DATA_BLOCK "InstGetSinaStatus"   // DB15
AUTHOR : Siemens Digital Industries
FAMILY : LAF
NAME : LAF_GetSinaStatus
VERSION : 1.1
// stored: InstanceOfName LAF_GetSinaStatus, InstanceOfType FB
"LAF_GetSinaStatus"
   // VAR_INPUT
   //    enable : Bool;
   // END_VAR
   // VAR_OUTPUT
   //    valid { ExternalWritable := 'False'} : Bool;
   //    busy { ExternalWritable := 'False'} : Bool;
   //    error { ExternalWritable := 'False'} : Bool;
   //    status { ExternalWritable := 'False'} : Word;
   //    diagnostics { ExternalWritable := 'False'} : "LAF_typeDiagnostics";
   //    statusWriteRecord { ExternalVisible := 'False'; ExternalWritable := 'False'} : DWord;
   //    statusReadRecord { ExternalWritable := 'False'} : DWord;
   // END_VAR
   // VAR_IN_OUT
   //    configuration : Array[*] of "LAF_typeDriveDiagConfig";
   //    moduleInterface : "LAF_typeDriveDiagInterfaceHmi";
   // END_VAR
   // VAR
   //    statInternal { ExternalAccessible := 'False'; ExternalVisible := 'False'; ExternalWritable := 'False'} : Struct
   //       enablePrevious : Bool;
   //       valid : Bool;
   //       busy : Bool;
   //       error : Bool;
   //       errorUserCleared : Bool;
   //       errorAutoCleared : Bool;
   //       disablingCompleted : Bool;
   //       diagnostics : "LAF_typeDiagnostics";
   //       emptyDiagnostics : "LAF_typeDiagnostics";
   //    END_STRUCT;
   //    statMainState { ExternalAccessible := 'False'; ExternalVisible := 'False'; ExternalWritable := 'False'} : DInt;
   //    statArrayMin { ExternalAccessible := 'False'; ExternalVisible := 'False'; ExternalWritable := 'False'} : DInt;
   //    statArrayMax { ExternalAccessible := 'False'; ExternalVisible := 'False'; ExternalWritable := 'False'} : DInt;
   //    instWriteRecord { ExternalAccessible := 'False'; ExternalVisible := 'False'; ExternalWritable := 'False'} : WRREC;
   //    instReadRecord { ExternalAccessible := 'False'; ExternalVisible := 'False'; ExternalWritable := 'False'} : RDREC;
   //    statWriteReq { ExternalAccessible := 'False'; ExternalVisible := 'False'; ExternalWritable := 'False'} : Struct
   //       header : Struct
   //          reqRef : Byte;
   //          reqID : Byte;
   //          axis : Byte;
   //          noPara : Byte;
   //       END_STRUCT;
   //       data : Array[0..235] of Byte;
   //    END_STRUCT;
   //    statReadReq { ExternalAccessible := 'False'; ExternalVisible := 'False'; ExternalWritable := 'False'} : Struct
   //       header : Struct
   //          reqRef : Byte;
   //          reqID : Byte;
   //          axis : Byte;
   //          noPara : Byte;
   //       END_STRUCT;
   //       data : Array[0..235] of Byte;
   //    END_STRUCT;
   //    instActTimer { ExternalAccessible := 'False'; ExternalVisible := 'False'; ExternalWritable := 'False'} : IEC_TIMER;
   //    instReqTimer { ExternalAccessible := 'False'; ExternalVisible := 'False'; ExternalWritable := 'False'} : IEC_TIMER;
   //    statDataTransRun { ExternalAccessible := 'False'; ExternalVisible := 'False'; ExternalWritable := 'False'} : Bool;
   //    statWriteReqSet { ExternalAccessible := 'False'; ExternalVisible := 'False'; ExternalWritable := 'False'} : Bool;
   //    statActTimerIn { ExternalAccessible := 'False'; ExternalVisible := 'False'; ExternalWritable := 'False'} : Bool;
   //    statPrevTimeValue { ExternalAccessible := 'False'; ExternalVisible := 'False'; ExternalWritable := 'False'} : Time;
   //    statActTimerValueAct { ExternalAccessible := 'False'; ExternalVisible := 'False'; ExternalWritable := 'False'} : Time;
   //    statActTimerValueReq { ExternalAccessible := 'False'; ExternalVisible := 'False'; ExternalWritable := 'False'} : Time;
   //    statPrevDriveIndex { ExternalAccessible := 'False'; ExternalVisible := 'False'; ExternalWritable := 'False'} : DInt;
   // END_VAR
BEGIN
END_DATA_BLOCK

DATA_BLOCK "InstInterfaceSignals"   // DB39
{ DB_Accessible_From_OPC_UA := 'FALSE' }
AUTHOR : SICAR
FAMILY : Diag
VERSION : 1.0
// stored: DBAccessibleFromOPCUA false, DBAccessibleFromWebserver false, InstanceOfName CallInterfaceSignals, InstanceOfType FB
"CallInterfaceSignals"
BEGIN
   statInterfaceSignalsHmi[1].valueSymbolLeft.freeDescriptionText := WSTRING#'ReelCut To STK30';
   statInterfaceSignalsHmi[2].valueSymbolLeft.freeDescriptionText := WSTRING#'ReelCut to STK40';
   statInterfaceSignalsHmi[3].valueSymbolLeft.freeDescriptionText := WSTRING#'BK01';
   statInterfaceSignalsHmi[4].valueSymbolLeft.freeDescriptionText := WSTRING#'BK02';
   statInterfaceSignalsHmi[5].valueSymbolLeft.freeDescriptionText := WSTRING#'BK03';
   statInterfaceSignalsHmi[6].valueSymbolLeft.freeDescriptionText := WSTRING#'BK04';
   statInterfaceSignalsHmi[7].valueSymbolLeft.freeDescriptionText := WSTRING#'BK05';
   statInterfaceSignalsHmi[8].valueSymbolLeft.freeDescriptionText := WSTRING#'BK06';
   statInterfaceSignalsHmi[9].valueSymbolLeft.freeDescriptionText := WSTRING#'BK07';
   statInterfaceSignalsHmi[10].valueSymbolLeft.freeDescriptionText := WSTRING#'BK08';
   statInterfaceSignalsHmi[11].valueSymbolLeft.freeDescriptionText := WSTRING#'BK09';
   statInterfaceSignalsHmi[12].valueSymbolLeft.freeDescriptionText := WSTRING#'BK10';
   statInterfaceSignalsHmi[13].valueSymbolLeft.freeDescriptionText := WSTRING#'SBK01';
   statInterfaceSignalsHmi[14].valueSymbolLeft.freeDescriptionText := WSTRING#'SBK02';
   statInterfaceSignalsHmi[15].valueSymbolLeft.freeDescriptionText := WSTRING#'SBK03';
   statInterfaceSignalsHmi[16].valueSymbolLeft.freeDescriptionText := WSTRING#'SBK04';
   statInterfaceSignalsHmi[17].valueSymbolLeft.freeDescriptionText := WSTRING#'SBK05';
   statInterfaceSignalsHmi[18].valueSymbolLeft.freeDescriptionText := WSTRING#'SBK06';
   statInterfaceSignalsHmi[19].valueSymbolLeft.freeDescriptionText := WSTRING#'SBK01';
   statInterfaceSignalsHmi[20].valueSymbolLeft.freeDescriptionText := WSTRING#'SBK02';
   statInterfaceSignalsHmi[21].valueSymbolLeft.freeDescriptionText := WSTRING#'SBK03';
   statInterfaceSignalsHmi[22].valueSymbolLeft.freeDescriptionText := WSTRING#'SBK04';
   statInterfaceSignalsHmi[23].valueSymbolLeft.freeDescriptionText := WSTRING#'SBK05';
   statInterfaceSignalsHmi[24].valueSymbolLeft.freeDescriptionText := WSTRING#'SBK06';
   statInterfaceSignalsHmi[25].valueSymbolLeft.freeDescriptionText := WSTRING#'SBK07';
   statInterfaceSignalsHmi[26].valueSymbolLeft.freeDescriptionText := WSTRING#'SBK08';
   statInterfaceSignalsHmi[27].valueSymbolLeft.freeDescriptionText := WSTRING#'SBK09';
   statInterfaceSignalsHmi[28].valueSymbolLeft.freeDescriptionText := WSTRING#'PM01';
   statInterfaceSignalsHmi[29].valueSymbolLeft.freeDescriptionText := WSTRING#'PM02';
   statInterfaceSignalsHmi[30].valueSymbolLeft.freeDescriptionText := WSTRING#'PM03';
   statInterfaceSignalsHmi[31].valueSymbolLeft.freeDescriptionText := WSTRING#'PM04';
   statInterfaceSignalsHmi[37].valueSymbolLeft.freeDescriptionText := WSTRING#'SP501';
   statInterfaceSignalsHmi[38].valueSymbolLeft.freeDescriptionText := WSTRING#'SP502';
   statInterfaceSignalsHmi[39].valueSymbolLeft.freeDescriptionText := WSTRING#'SP503';
   statInterfaceSignalsHmi[40].valueSymbolLeft.freeDescriptionText := WSTRING#'SP504';
   statInterfaceSignalsHmi[41].valueSymbolLeft.freeDescriptionText := WSTRING#'SP505';
   statInterfaceSignalsHmi[42].valueSymbolLeft.freeDescriptionText := WSTRING#'SP506';
   statInterfaceSignalsHmi[43].valueSymbolLeft.freeDescriptionText := WSTRING#'SP507';
   statInterfaceSignalsHmi[44].valueSymbolLeft.freeDescriptionText := WSTRING#'SP508';
   statInterfaceSignalsHmi[45].valueSymbolLeft.freeDescriptionText := WSTRING#'SP509';
   statInterfaceSignalsHmi[46].valueSymbolLeft.freeDescriptionText := WSTRING#'SP510';
   statInterfaceSignalsHmi[47].valueSymbolLeft.freeDescriptionText := WSTRING#'SP511';
   statInterfaceSignalsHmi[48].valueSymbolLeft.freeDescriptionText := WSTRING#'SP512';
   statInterfaceSignalsHmi[1].valueSymbolRight.freeDescriptionText := WSTRING#'ReelCut To STK30';
   statInterfaceSignalsHmi[2].valueSymbolRight.freeDescriptionText := WSTRING#'ReelCut to STK40';
   statInterfaceSignalsHmi[3].valueSymbolRight.freeDescriptionText := WSTRING#'BK01';
   statInterfaceSignalsHmi[4].valueSymbolRight.freeDescriptionText := WSTRING#'BK02';
   statInterfaceSignalsHmi[5].valueSymbolRight.freeDescriptionText := WSTRING#'BK03';
   statInterfaceSignalsHmi[6].valueSymbolRight.freeDescriptionText := WSTRING#'BK04';
   statInterfaceSignalsHmi[7].valueSymbolRight.freeDescriptionText := WSTRING#'BK05';
   statInterfaceSignalsHmi[8].valueSymbolRight.freeDescriptionText := WSTRING#'BK06';
   statInterfaceSignalsHmi[9].valueSymbolRight.freeDescriptionText := WSTRING#'BK07';
   statInterfaceSignalsHmi[10].valueSymbolRight.freeDescriptionText := WSTRING#'BK08';
   statInterfaceSignalsHmi[11].valueSymbolRight.freeDescriptionText := WSTRING#'BK09';
   statInterfaceSignalsHmi[12].valueSymbolRight.freeDescriptionText := WSTRING#'BK10';
   statInterfaceSignalsHmi[13].valueSymbolRight.freeDescriptionText := WSTRING#'SBK01';
   statInterfaceSignalsHmi[14].valueSymbolRight.freeDescriptionText := WSTRING#'SBK02';
   statInterfaceSignalsHmi[15].valueSymbolRight.freeDescriptionText := WSTRING#'SBK03';
   statInterfaceSignalsHmi[16].valueSymbolRight.freeDescriptionText := WSTRING#'SBK04';
   statInterfaceSignalsHmi[17].valueSymbolRight.freeDescriptionText := WSTRING#'SBK05';
   statInterfaceSignalsHmi[18].valueSymbolRight.freeDescriptionText := WSTRING#'SBK06';
   statInterfaceSignalsHmi[19].valueSymbolRight.freeDescriptionText := WSTRING#'SBK01';
   statInterfaceSignalsHmi[20].valueSymbolRight.freeDescriptionText := WSTRING#'SBK02';
   statInterfaceSignalsHmi[21].valueSymbolRight.freeDescriptionText := WSTRING#'SBK03';
   statInterfaceSignalsHmi[22].valueSymbolRight.freeDescriptionText := WSTRING#'SBK04';
   statInterfaceSignalsHmi[23].valueSymbolRight.freeDescriptionText := WSTRING#'SBK05';
   statInterfaceSignalsHmi[24].valueSymbolRight.freeDescriptionText := WSTRING#'SBK06';
   statInterfaceSignalsHmi[25].valueSymbolRight.freeDescriptionText := WSTRING#'SBK07';
   statInterfaceSignalsHmi[26].valueSymbolRight.freeDescriptionText := WSTRING#'SBK08';
   statInterfaceSignalsHmi[27].valueSymbolRight.freeDescriptionText := WSTRING#'SBK09';
   statInterfaceSignalsHmi[28].valueSymbolRight.freeDescriptionText := WSTRING#'PM01';
   statInterfaceSignalsHmi[29].valueSymbolRight.freeDescriptionText := WSTRING#'PM02';
   statInterfaceSignalsHmi[30].valueSymbolRight.freeDescriptionText := WSTRING#'PM03';
   statInterfaceSignalsHmi[31].valueSymbolRight.freeDescriptionText := WSTRING#'PM04';
   statInterfaceSignalsHmi[37].valueSymbolRight.freeDescriptionText := WSTRING#'SP501';
   statInterfaceSignalsHmi[38].valueSymbolRight.freeDescriptionText := WSTRING#'SP502';
   statInterfaceSignalsHmi[39].valueSymbolRight.freeDescriptionText := WSTRING#'SP503';
   statInterfaceSignalsHmi[40].valueSymbolRight.freeDescriptionText := WSTRING#'SP504';
   statInterfaceSignalsHmi[41].valueSymbolRight.freeDescriptionText := WSTRING#'SP505';
   statInterfaceSignalsHmi[42].valueSymbolRight.freeDescriptionText := WSTRING#'SP506';
   statInterfaceSignalsHmi[43].valueSymbolRight.freeDescriptionText := WSTRING#'SP507';
   statInterfaceSignalsHmi[44].valueSymbolRight.freeDescriptionText := WSTRING#'SP508';
   statInterfaceSignalsHmi[45].valueSymbolRight.freeDescriptionText := WSTRING#'SP509';
   statInterfaceSignalsHmi[46].valueSymbolRight.freeDescriptionText := WSTRING#'SP510';
   statInterfaceSignalsHmi[47].valueSymbolRight.freeDescriptionText := WSTRING#'SP511';
   statInterfaceSignalsHmi[48].valueSymbolRight.freeDescriptionText := WSTRING#'SP512';
END_DATA_BLOCK

DATA_BLOCK "InstInterfaceSignalsConv_BA30"   // DB59
// stored: InstanceOfName CallInterfaceSignalsConv, InstanceOfType FB
"CallInterfaceSignalsConv"
BEGIN
END_DATA_BLOCK

DATA_BLOCK "InstInterfaceSignalsConv_BA40"   // DB136
// stored: InstanceOfName CallInterfaceSignalsConv, InstanceOfType FB
"CallInterfaceSignalsConv"
BEGIN
END_DATA_BLOCK

DATA_BLOCK "InstProfinetDeviceDiagStatus"   // DB172
// stored: InstanceOfName LER_DiagnosticsStatus, InstanceOfType FB
"LER_DiagnosticsStatus"
   // VAR_INPUT
   //    devStateHmi_X1 : Array[0..256] of "LAF_typeDevDiagBasic";
   //    devStateHmi_X2 : Array[0..256] of "LAF_typeDevDiagBasic";
   //    UnitSelect : Int;
   //    Reset : Bool;
   // END_VAR
   // VAR_IN_OUT
   //    DevState : "LER_DiagnosticsInterface";
   // END_VAR
   // VAR
   //    staticCntState : Int;
   //    staticCntStartState : Int;
   //    staticCntEndState : Int;
   //    staticCntDev : Int;
   //    staticCntHighLimit_X2 : Array[1..15] of Int;
   //    staticCntLowLimit_X2 : Array[1..15] of Int;
   //    staticCntHighLimit_X1 : Array[1..15] of Int;
   //    staticCntLowLimit_X1 : Array[1..15] of Int;
   //    staticCntModuleState : Int;
   //    staticDevStateError : Array[0..15] of Bool;
   //    statiDevStateMove_X1 : Array[0..15] of Int;
   //    statiDevStateMove_X2 : Array[0..15] of Int;
   // END_VAR
BEGIN
END_DATA_BLOCK

DATA_BLOCK "InstProfinetDeviceDiag_x1"   // DB174
AUTHOR : Siemens Digital Industries
FAMILY : LAF
// stored: AssignedProDiagFB ProDiag, InstanceOfName LAF_ProfinetDevDiag, InstanceOfType FB
"LAF_ProfinetDevDiag"
   // VAR_INPUT
   //    plantIdentifier { ExternalAccessible := 'False'; ExternalVisible := 'False'; ExternalWritable := 'False'} : WString[24];
   //    textListId { ExternalAccessible := 'False'; ExternalVisible := 'False'; ExternalWritable := 'False'} : Int;
   //    localProfinetSystem { ExternalAccessible := 'False'; ExternalVisible := 'False'; ExternalWritable := 'False'} : HW_IOSYSTEM;
   //    firstCycle { ExternalAccessible := 'False'; ExternalVisible := 'False'; ExternalWritable := 'False'} : Bool;
   //    maxDevicesDiag { ExternalAccessible := 'False'; ExternalVisible := 'False'; ExternalWritable := 'False'} : DInt;
   //    maxModulesDiag { ExternalAccessible := 'False'; ExternalVisible := 'False'; ExternalWritable := 'False'} : DInt;
   //    ackAlarms { ExternalAccessible := 'False'; ExternalVisible := 'False'; ExternalWritable := 'False'} : Bool;
   //    hideAlarmMask { ExternalAccessible := 'False'; ExternalVisible := 'False'; ExternalWritable := 'False'} : Word;
   // END_VAR
   // VAR_OUTPUT
   //    generalAlarm { ExternalAccessible := 'False'; ExternalVisible := 'False'; ExternalWritable := 'False'} : Bool;
   //    deviceFaulty { ExternalAccessible := 'False'; ExternalVisible := 'False'; ExternalWritable := 'False'} : Bool;
   //    deviceProblem { ExternalAccessible := 'False'; ExternalVisible := 'False'; ExternalWritable := 'False'} : Bool;
   //    deviceDeactivated { ExternalAccessible := 'False'; ExternalVisible := 'False'; ExternalWritable := 'False'} : Bool;
   //    deviceNotPresent { ExternalAccessible := 'False'; ExternalVisible := 'False'; ExternalWritable := 'False'} : Bool;
   // END_VAR
   // VAR_IN_OUT
   //    interfaceDevDiag : "LAF_typeDevDiagInterface";
   // END_VAR
   // VAR
   //    statDevDiagInternal { ExternalAccessible := 'False'; ExternalVisible := 'False'; ExternalWritable := 'False'} : "LAF_typeDevDiagInternal";
   //    statCnt1ShotGetName { ExternalAccessible := 'False'; ExternalVisible := 'False'; ExternalWritable := 'False'} : DInt;
   //    statCnt1ShotGeo2Log { ExternalAccessible := 'False'; ExternalVisible := 'False'; ExternalWritable := 'False'} : DInt;
   //    statCnt1ShotGetImDat { ExternalAccessible := 'False'; ExternalVisible := 'False'; ExternalWritable := 'False'} : DInt;
   //    statCntCyclDevState { ExternalAccessible := 'False'; ExternalVisible := 'False'; ExternalWritable := 'False'} : DInt;
   //    statCntCyclState { ExternalAccessible := 'False'; ExternalVisible := 'False'; ExternalWritable := 'False'} : DInt;
   //    statCntCyclModulState { ExternalAccessible := 'False'; ExternalVisible := 'False'; ExternalWritable := 'False'} : DInt;
   //    statCntCyclGetDiag { ExternalAccessible := 'False'; ExternalVisible := 'False'; ExternalWritable := 'False'} : DInt;
   //    statBusy { ExternalAccessible := 'False'; ExternalVisible := 'False'; ExternalWritable := 'False'} : "LAF_typeDevDiagStateInstruct";
   //    statDone { ExternalAccessible := 'False'; ExternalVisible := 'False'; ExternalWritable := 'False'} : "LAF_typeDevDiagStateInstruct";
   //    statOtherInstruct { ExternalAccessible := 'False'; ExternalVisible := 'False'; ExternalWritable := 'False'} : "LAF_typeDevDiagInstruct";
   //    instGetName { ExternalAccessible := 'False'; ExternalVisible := 'False'; ExternalWritable := 'False'} : Get_Name;
   //    statGetNameDat { ExternalAccessible := 'False'; ExternalVisible := 'False'; ExternalWritable := 'False'} : String[24];
   //    statGetNameErrorStatus { ExternalAccessible := 'False'; ExternalVisible := 'False'; ExternalWritable := 'False'} : Word;
   //    statGetNameErrorDevCycle { ExternalAccessible := 'False'; ExternalVisible := 'False'; ExternalWritable := 'False'} : DInt;
   //    instGetImData { ExternalAccessible := 'False'; ExternalVisible := 'False'; ExternalWritable := 'False'} : Get_IM_Data;
   //    statIm0Data { ExternalAccessible := 'False'; ExternalVisible := 'False'; ExternalWritable := 'False'} : IM0_Data;
   //    statGetImDatErrorStatus { ExternalAccessible := 'False'; ExternalVisible := 'False'; ExternalWritable := 'False'} : Word;
   //    statGetImDatErrorCycle { ExternalAccessible := 'False'; ExternalVisible := 'False'; ExternalWritable := 'False'} : DInt;
   //    statAlarm { ExternalAccessible := 'False'; ExternalVisible := 'False'; ExternalWritable := 'False'} : "LAF_typeDevDiagAlarm";
   //    statHideAlarm { ExternalAccessible := 'False'; ExternalVisible := 'False'; ExternalWritable := 'False'} : "LAF_typeDevDiagAlarm";
   //    statRisPushbutton { ExternalAccessible := 'False'; ExternalVisible := 'False'; ExternalWritable := 'False'} : "LAF_typeDevDiagRisEdge";
   //    statErrorText { ExternalAccessible := 'False'; ExternalVisible := 'False'; ExternalWritable := 'False'} : String[24];
   //    stat8CharError { ExternalAccessible := 'False'; ExternalVisible := 'False'; ExternalWritable := 'False'} : String[8];
   //    statAlarmNo { ExternalAccessible := 'False'; ExternalVisible := 'False'; ExternalWritable := 'False'} : Array[0..23] of UInt;
   // END_VAR
BEGIN
END_DATA_BLOCK

DATA_BLOCK "InstProfinetDeviceDiag_x2"   // DB170
AUTHOR : Siemens Digital Industries
FAMILY : LAF
VERSION : 1.2
// stored: AssignedProDiagFB ProDiag, InstanceOfName LAF_ProfinetDevDiag, InstanceOfType FB
"LAF_ProfinetDevDiag"
   // VAR_INPUT
   //    plantIdentifier { ExternalAccessible := 'False'; ExternalVisible := 'False'; ExternalWritable := 'False'} : WString[24];
   //    textListId { ExternalAccessible := 'False'; ExternalVisible := 'False'; ExternalWritable := 'False'} : Int;
   //    localProfinetSystem { ExternalAccessible := 'False'; ExternalVisible := 'False'; ExternalWritable := 'False'} : HW_IOSYSTEM;
   //    firstCycle { ExternalAccessible := 'False'; ExternalVisible := 'False'; ExternalWritable := 'False'} : Bool;
   //    maxDevicesDiag { ExternalAccessible := 'False'; ExternalVisible := 'False'; ExternalWritable := 'False'} : DInt;
   //    maxModulesDiag { ExternalAccessible := 'False'; ExternalVisible := 'False'; ExternalWritable := 'False'} : DInt;
   //    ackAlarms { ExternalAccessible := 'False'; ExternalVisible := 'False'; ExternalWritable := 'False'} : Bool;
   //    hideAlarmMask { ExternalAccessible := 'False'; ExternalVisible := 'False'; ExternalWritable := 'False'} : Word;
   // END_VAR
   // VAR_OUTPUT
   //    generalAlarm { ExternalAccessible := 'False'; ExternalVisible := 'False'; ExternalWritable := 'False'} : Bool;
   //    deviceFaulty { ExternalAccessible := 'False'; ExternalVisible := 'False'; ExternalWritable := 'False'} : Bool;
   //    deviceProblem { ExternalAccessible := 'False'; ExternalVisible := 'False'; ExternalWritable := 'False'} : Bool;
   //    deviceDeactivated { ExternalAccessible := 'False'; ExternalVisible := 'False'; ExternalWritable := 'False'} : Bool;
   //    deviceNotPresent { ExternalAccessible := 'False'; ExternalVisible := 'False'; ExternalWritable := 'False'} : Bool;
   // END_VAR
   // VAR_IN_OUT
   //    interfaceDevDiag : "LAF_typeDevDiagInterface";
   // END_VAR
   // VAR
   //    statDevDiagInternal { ExternalAccessible := 'False'; ExternalVisible := 'False'; ExternalWritable := 'False'} : "LAF_typeDevDiagInternal";
   //    statCnt1ShotGetName { ExternalAccessible := 'False'; ExternalVisible := 'False'; ExternalWritable := 'False'} : DInt;
   //    statCnt1ShotGeo2Log { ExternalAccessible := 'False'; ExternalVisible := 'False'; ExternalWritable := 'False'} : DInt;
   //    statCnt1ShotGetImDat { ExternalAccessible := 'False'; ExternalVisible := 'False'; ExternalWritable := 'False'} : DInt;
   //    statCntCyclDevState { ExternalAccessible := 'False'; ExternalVisible := 'False'; ExternalWritable := 'False'} : DInt;
   //    statCntCyclState { ExternalAccessible := 'False'; ExternalVisible := 'False'; ExternalWritable := 'False'} : DInt;
   //    statCntCyclModulState { ExternalAccessible := 'False'; ExternalVisible := 'False'; ExternalWritable := 'False'} : DInt;
   //    statCntCyclGetDiag { ExternalAccessible := 'False'; ExternalVisible := 'False'; ExternalWritable := 'False'} : DInt;
   //    statBusy { ExternalAccessible := 'False'; ExternalVisible := 'False'; ExternalWritable := 'False'} : "LAF_typeDevDiagStateInstruct";
   //    statDone { ExternalAccessible := 'False'; ExternalVisible := 'False'; ExternalWritable := 'False'} : "LAF_typeDevDiagStateInstruct";
   //    statOtherInstruct { ExternalAccessible := 'False'; ExternalVisible := 'False'; ExternalWritable := 'False'} : "LAF_typeDevDiagInstruct";
   //    instGetName { ExternalAccessible := 'False'; ExternalVisible := 'False'; ExternalWritable := 'False'} : Get_Name;
   //    statGetNameDat { ExternalAccessible := 'False'; ExternalVisible := 'False'; ExternalWritable := 'False'} : String[24];
   //    statGetNameErrorStatus { ExternalAccessible := 'False'; ExternalVisible := 'False'; ExternalWritable := 'False'} : Word;
   //    statGetNameErrorDevCycle { ExternalAccessible := 'False'; ExternalVisible := 'False'; ExternalWritable := 'False'} : DInt;
   //    instGetImData { ExternalAccessible := 'False'; ExternalVisible := 'False'; ExternalWritable := 'False'} : Get_IM_Data;
   //    statIm0Data { ExternalAccessible := 'False'; ExternalVisible := 'False'; ExternalWritable := 'False'} : IM0_Data;
   //    statGetImDatErrorStatus { ExternalAccessible := 'False'; ExternalVisible := 'False'; ExternalWritable := 'False'} : Word;
   //    statGetImDatErrorCycle { ExternalAccessible := 'False'; ExternalVisible := 'False'; ExternalWritable := 'False'} : DInt;
   //    statAlarm { ExternalAccessible := 'False'; ExternalVisible := 'False'; ExternalWritable := 'False'} : "LAF_typeDevDiagAlarm";
   //    statHideAlarm { ExternalAccessible := 'False'; ExternalVisible := 'False'; ExternalWritable := 'False'} : "LAF_typeDevDiagAlarm";
   //    statRisPushbutton { ExternalAccessible := 'False'; ExternalVisible := 'False'; ExternalWritable := 'False'} : "LAF_typeDevDiagRisEdge";
   //    statErrorText { ExternalAccessible := 'False'; ExternalVisible := 'False'; ExternalWritable := 'False'} : String[24];
   //    stat8CharError { ExternalAccessible := 'False'; ExternalVisible := 'False'; ExternalWritable := 'False'} : String[8];
   //    statAlarmNo { ExternalAccessible := 'False'; ExternalVisible := 'False'; ExternalWritable := 'False'} : Array[0..23] of UInt;
   // END_VAR
BEGIN
END_DATA_BLOCK

DATA_BLOCK "ReelCutToStack30"   // DB184
// stored: InstanceOfName typeReelCutToStack, InstanceOfType UDT
"typeReelCutToStack"
BEGIN
END_DATA_BLOCK

DATA_BLOCK "ReelCutToStack40"   // DB223
// stored: InstanceOfName typeReelCutToStack, InstanceOfType UDT
"typeReelCutToStack"
BEGIN
END_DATA_BLOCK

DATA_BLOCK "StackToReelCut30"   // DB185
// stored: InstanceOfName typeStackToReelCut, InstanceOfType UDT
"typeStackToReelCut"
BEGIN
END_DATA_BLOCK

DATA_BLOCK "StackToReelCut40"   // DB224
// stored: InstanceOfName typeStackToReelCut, InstanceOfType UDT
"typeStackToReelCut"
BEGIN
END_DATA_BLOCK

DATA_BLOCK "PNDevDiagInterface_X1"   // DB261
// stored: InstanceOfName LAF_typeDevDiagInterface, InstanceOfType UDT
"LAF_typeDevDiagInterface"
   // VAR
   //    globalInfoHmi : "LAF_typeDevDiagGlobal";
   //    devStateHmi { ExternalWritable := 'False'} : Array[0..256] of "LAF_typeDevDiagBasic";
   //    devStateUser { ExternalAccessible := 'False'; ExternalVisible := 'False'; ExternalWritable := 'False'} : Array[0..256] of "LAF_typeDevDiagState";
   // END_VAR
BEGIN
END_DATA_BLOCK

DATA_BLOCK "PNDevDiagInterface_X2"   // DB48
// stored: InstanceOfName LAF_typeDevDiagInterface, InstanceOfType UDT
"LAF_typeDevDiagInterface"
   // VAR
   //    globalInfoHmi : "LAF_typeDevDiagGlobal";
   //    devStateHmi { ExternalWritable := 'False'} : Array[0..256] of "LAF_typeDevDiagBasic";
   //    devStateUser { ExternalAccessible := 'False'; ExternalVisible := 'False'; ExternalWritable := 'False'} : Array[0..256] of "LAF_typeDevDiagState";
   // END_VAR
BEGIN
END_DATA_BLOCK

DATA_BLOCK "PNDevDiagStatus"   // DB173
// stored: InstanceOfName LER_DiagnosticsInterface, InstanceOfType UDT
"LER_DiagnosticsInterface"
   // VAR
   //    DevState { S7_SetPoint := 'True'} : "LER_DevState";
   //    DigState { S7_SetPoint := 'True'} : Array[0..15] of Bool;
   //    Station_Position : Int;
   // END_VAR
BEGIN
END_DATA_BLOCK

DATA_BLOCK "instZa_TraceCodeGenerationLeft"   // DB226
// stored: InstanceOfName za_TraceCodeGeneration, InstanceOfType FB
"za_TraceCodeGeneration"
   // VAR_INPUT
   //    ComponentType : String;
   //    MfgSiteId : String;
   //    Shift : String;
   //    LineIdentifier : String;
   //    GMPartNumber : String;
   //    SignalForTC_Creation : Bool;
   //    SignalForSN_Increment : Bool;
   //    SignalForSN_Reset : Bool;
   //    SignalForTCBuffer_Clear : Bool;
   //    AlwaysON : Bool;
   //    ProgramID : String;
   //    System_Clock_1s_Pulse : Bool;
   // END_VAR
   // VAR_OUTPUT
   //    TracebilityCode : String;
   //    TracebilityCode_Ready : Bool;
   //    Tracecode : Array[1..20] of Char;
   //    PartNumber : Array[1..8] of Char;
   // END_VAR
   // VAR
   //    TCtimer : TON_TIME;
   // END_VAR
   // VAR RETAIN
   //    instCounter : CTU_DINT;
   //    statPrevTraceBilityCode : String;
   // END_VAR
   // VAR
   //    statPrevDailySequenceNumber : DInt;
   //    TraceCodeData { ExternalAccessible := 'False'; ExternalVisible := 'False'; ExternalWritable := 'False'} : Array[0..20] of String[26];
   //    TraceCellNumber { ExternalAccessible := 'False'; ExternalVisible := 'False'; ExternalWritable := 'False'} : Array[0..20] of USInt;
   //    statTracecodeBuffer : Array[1..20] of Char;
   //    statPartNumberBuffer : Array[1..8] of Char;
   //    statTracecodeBufferCnt : UInt;
   //    statPartNumberBufferCnt : UInt;
   // END_VAR
BEGIN
END_DATA_BLOCK

DATA_BLOCK "instZa_TraceCodeGenerationRight"   // DB232
// stored: InstanceOfName za_TraceCodeGeneration, InstanceOfType FB
"za_TraceCodeGeneration"
   // VAR_INPUT
   //    ComponentType : String;
   //    MfgSiteId : String;
   //    Shift : String;
   //    LineIdentifier : String;
   //    GMPartNumber : String;
   //    SignalForTC_Creation : Bool;
   //    SignalForSN_Increment : Bool;
   //    SignalForSN_Reset : Bool;
   //    SignalForTCBuffer_Clear : Bool;
   //    AlwaysON : Bool;
   //    ProgramID : String;
   //    System_Clock_1s_Pulse : Bool;
   // END_VAR
   // VAR_OUTPUT
   //    TracebilityCode : String;
   //    TracebilityCode_Ready : Bool;
   //    Tracecode : Array[1..20] of Char;
   //    PartNumber : Array[1..8] of Char;
   // END_VAR
   // VAR
   //    TCtimer : TON_TIME;
   // END_VAR
   // VAR RETAIN
   //    instCounter : CTU_DINT;
   //    statPrevTraceBilityCode : String;
   // END_VAR
   // VAR
   //    statPrevDailySequenceNumber : DInt;
   //    TraceCodeData { ExternalAccessible := 'False'; ExternalVisible := 'False'; ExternalWritable := 'False'} : Array[0..20] of String[26];
   //    TraceCellNumber { ExternalAccessible := 'False'; ExternalVisible := 'False'; ExternalWritable := 'False'} : Array[0..20] of USInt;
   //    statTracecodeBuffer : Array[1..20] of Char;
   //    statPartNumberBuffer : Array[1..8] of Char;
   //    statTracecodeBufferCnt : UInt;
   //    statPartNumberBufferCnt : UInt;
   // END_VAR
BEGIN
END_DATA_BLOCK

DATA_BLOCK "za_TraceCodeGeneration_DB"   // DB263
// stored: InstanceOfName za_TraceCodeGeneration, InstanceOfType FB
"za_TraceCodeGeneration"
   // VAR_INPUT
   //    ComponentType : String;
   //    MfgSiteId : String;
   //    Shift : String;
   //    LineIdentifier : String;
   //    GMPartNumber : String;
   //    SignalForTC_Creation : Bool;
   //    SignalForSN_Increment : Bool;
   //    SignalForSN_Reset : Bool;
   //    SignalForTCBuffer_Clear : Bool;
   //    AlwaysON : Bool;
   //    ProgramID : String;
   //    System_Clock_1s_Pulse : Bool;
   // END_VAR
   // VAR_OUTPUT
   //    TracebilityCode : String;
   //    TracebilityCode_Ready : Bool;
   //    Tracecode : Array[1..20] of Char;
   //    PartNumber : Array[1..8] of Char;
   // END_VAR
   // VAR
   //    TCtimer : TON_TIME;
   // END_VAR
   // VAR RETAIN
   //    instCounter : CTU_DINT;
   //    statPrevTraceBilityCode : String;
   // END_VAR
   // VAR
   //    statPrevDailySequenceNumber : DInt;
   //    TraceCodeData { ExternalAccessible := 'False'; ExternalVisible := 'False'; ExternalWritable := 'False'} : Array[0..20] of String[26];
   //    TraceCellNumber { ExternalAccessible := 'False'; ExternalVisible := 'False'; ExternalWritable := 'False'} : Array[0..20] of USInt;
   //    statTracecodeBuffer : Array[1..20] of Char;
   //    statPartNumberBuffer : Array[1..8] of Char;
   //    statTracecodeBufferCnt : UInt;
   //    statPartNumberBufferCnt : UInt;
   // END_VAR
BEGIN
END_DATA_BLOCK

DATA_BLOCK "InstCompValEqOr1"   // DB132
TITLE = Instanz CompValEqOr1 / Instance CompValEqOr1
{ DB_Accessible_From_OPC_UA := 'FALSE' }
AUTHOR : SICAR
FAMILY : Miscellaneous
VERSION : 1.0
// Instanz DB / Instance DB
// stored: DBAccessibleFromOPCUA false, InstanceOfName CompValEqOr, InstanceOfType FB
"CompValEqOr"
BEGIN
END_DATA_BLOCK

DATA_BLOCK "InstCompValEqOr2"   // DB133
TITLE = Instanz CompValEqOr2 / Instance CompValEqOr2
{ DB_Accessible_From_OPC_UA := 'FALSE' }
AUTHOR : SICAR
FAMILY : Miscellaneous
VERSION : 1.0
// Instanz DB / Instance DB
// stored: DBAccessibleFromOPCUA false, InstanceOfName CompValEqOr, InstanceOfType FB
"CompValEqOr"
BEGIN
END_DATA_BLOCK

DATA_BLOCK "InstCounterDataset1"   // DB65
TITLE = Instanz CounterDataset1 / Instance CounterDataset1
{ DB_Accessible_From_OPC_UA := 'FALSE' }
AUTHOR : SICAR
FAMILY : ProdData
// Instanz DB / Instance DB
// stored: DBAccessibleFromOPCUA false, InstanceOfName LSicar_ProdDataCounter, InstanceOfType FB
"LSicar_ProdDataCounter"
   // VAR_INPUT
   //    numberConfigDataSets { ExternalAccessible := 'False'; ExternalVisible := 'False'; ExternalWritable := 'False'} : Int;
   //    dataSetNumber { ExternalAccessible := 'False'; ExternalVisible := 'False'; ExternalWritable := 'False'} : UInt;
   // END_VAR
   // VAR_IN_OUT
   //    numberOfDataSets : "LSicar_typeNumberOfDataSets";
   //    dataSet : "LSicar_typeCounter";
   // END_VAR
   // VAR
   //    statCounter { ExternalAccessible := 'False'; ExternalVisible := 'False'; ExternalWritable := 'False'} : Array[0..20] of "LSicar_typeEdgePulseStruct";
   //    statRisEdgeResetAllExt { ExternalAccessible := 'False'; ExternalVisible := 'False'; ExternalWritable := 'False'} : Bool;
   //    statPosPulseResetAllExt { ExternalAccessible := 'False'; ExternalVisible := 'False'; ExternalWritable := 'False'} : Bool;
   //    statRisEdgeResetAll { ExternalAccessible := 'False'; ExternalVisible := 'False'; ExternalWritable := 'False'} : Bool;
   //    statPosPulseResetAll { ExternalAccessible := 'False'; ExternalVisible := 'False'; ExternalWritable := 'False'} : Bool;
   // END_VAR
BEGIN
END_DATA_BLOCK

DATA_BLOCK "InstCounterDataset2"   // DB66
TITLE = Instanz CounterDataSet2 / Instance CounterDataSet2
{ DB_Accessible_From_OPC_UA := 'FALSE' }
AUTHOR : SICAR
FAMILY : ProdData
// Instanz DB / Instance DB
// stored: DBAccessibleFromOPCUA false, InstanceOfName LSicar_ProdDataCounter, InstanceOfType FB
"LSicar_ProdDataCounter"
   // VAR_INPUT
   //    numberConfigDataSets { ExternalAccessible := 'False'; ExternalVisible := 'False'; ExternalWritable := 'False'} : Int;
   //    dataSetNumber { ExternalAccessible := 'False'; ExternalVisible := 'False'; ExternalWritable := 'False'} : UInt;
   // END_VAR
   // VAR_IN_OUT
   //    numberOfDataSets : "LSicar_typeNumberOfDataSets";
   //    dataSet : "LSicar_typeCounter";
   // END_VAR
   // VAR
   //    statCounter { ExternalAccessible := 'False'; ExternalVisible := 'False'; ExternalWritable := 'False'} : Array[0..20] of "LSicar_typeEdgePulseStruct";
   //    statRisEdgeResetAllExt { ExternalAccessible := 'False'; ExternalVisible := 'False'; ExternalWritable := 'False'} : Bool;
   //    statPosPulseResetAllExt { ExternalAccessible := 'False'; ExternalVisible := 'False'; ExternalWritable := 'False'} : Bool;
   //    statRisEdgeResetAll { ExternalAccessible := 'False'; ExternalVisible := 'False'; ExternalWritable := 'False'} : Bool;
   //    statPosPulseResetAll { ExternalAccessible := 'False'; ExternalVisible := 'False'; ExternalWritable := 'False'} : Bool;
   // END_VAR
BEGIN
END_DATA_BLOCK

DATA_BLOCK "InstCycleTimerDataset1"   // DB63
TITLE = Instanz CycleTimerDataset1 / Instance CycleTimerDataset1
{ DB_Accessible_From_OPC_UA := 'FALSE' }
AUTHOR : SICAR
FAMILY : ProdData
// Instanz DB / Instance DB
// stored: DBAccessibleFromOPCUA false, InstanceOfName LSicar_ProdDataCycleTimer, InstanceOfType FB
"LSicar_ProdDataCycleTimer"
   // VAR_INPUT
   //    numberConfigDataSets { ExternalAccessible := 'False'; ExternalVisible := 'False'; ExternalWritable := 'False'} : Int;
   //    dataSetNumber { ExternalAccessible := 'False'; ExternalVisible := 'False'; ExternalWritable := 'False'} : UInt;
   //    pulse100ms { ExternalAccessible := 'False'; ExternalVisible := 'False'; ExternalWritable := 'False'} : Bool;
   // END_VAR
   // VAR_IN_OUT
   //    numberOfDataSets : "LSicar_typeNumberOfDataSets";
   //    dataSet : "LSicar_typeCycleTimer";
   // END_VAR
   // VAR
   //    statCycleTimer { ExternalAccessible := 'False'; ExternalVisible := 'False'; ExternalWritable := 'False'} : Array[0..20] of "LSicar_typeCycleTimerStruct";
   //    statRisEdgeResetAllExt { ExternalAccessible := 'False'; ExternalVisible := 'False'; ExternalWritable := 'False'} : Bool;
   //    statPosPulseResetAllExt { ExternalAccessible := 'False'; ExternalVisible := 'False'; ExternalWritable := 'False'} : Bool;
   //    statRisEdgeResetAll { ExternalAccessible := 'False'; ExternalVisible := 'False'; ExternalWritable := 'False'} : Bool;
   //    statPosPulseResetAll { ExternalAccessible := 'False'; ExternalVisible := 'False'; ExternalWritable := 'False'} : Bool;
   // END_VAR
BEGIN
END_DATA_BLOCK

DATA_BLOCK "InstCycleTimerDataset2"   // DB79
TITLE = Instanz CycleTimerDataset2 / Instance CycleTimerDataset2
{ DB_Accessible_From_OPC_UA := 'FALSE' }
AUTHOR : SICAR
FAMILY : ProdData
// Instanz DB / Instance DB
// stored: DBAccessibleFromOPCUA false, InstanceOfName LSicar_ProdDataCycleTimer, InstanceOfType FB
"LSicar_ProdDataCycleTimer"
   // VAR_INPUT
   //    numberConfigDataSets { ExternalAccessible := 'False'; ExternalVisible := 'False'; ExternalWritable := 'False'} : Int;
   //    dataSetNumber { ExternalAccessible := 'False'; ExternalVisible := 'False'; ExternalWritable := 'False'} : UInt;
   //    pulse100ms { ExternalAccessible := 'False'; ExternalVisible := 'False'; ExternalWritable := 'False'} : Bool;
   // END_VAR
   // VAR_IN_OUT
   //    numberOfDataSets : "LSicar_typeNumberOfDataSets";
   //    dataSet : "LSicar_typeCycleTimer";
   // END_VAR
   // VAR
   //    statCycleTimer { ExternalAccessible := 'False'; ExternalVisible := 'False'; ExternalWritable := 'False'} : Array[0..20] of "LSicar_typeCycleTimerStruct";
   //    statRisEdgeResetAllExt { ExternalAccessible := 'False'; ExternalVisible := 'False'; ExternalWritable := 'False'} : Bool;
   //    statPosPulseResetAllExt { ExternalAccessible := 'False'; ExternalVisible := 'False'; ExternalWritable := 'False'} : Bool;
   //    statRisEdgeResetAll { ExternalAccessible := 'False'; ExternalVisible := 'False'; ExternalWritable := 'False'} : Bool;
   //    statPosPulseResetAll { ExternalAccessible := 'False'; ExternalVisible := 'False'; ExternalWritable := 'False'} : Bool;
   // END_VAR
BEGIN
END_DATA_BLOCK

DATA_BLOCK "InstCycleTimerDataset3"   // DB178
TITLE = Instanz CycleTimerDataset2 / Instance CycleTimerDataset2
{ DB_Accessible_From_OPC_UA := 'FALSE' }
AUTHOR : SICAR
FAMILY : ProdData
// Instanz DB / Instance DB
// stored: DBAccessibleFromOPCUA false, InstanceOfName LSicar_ProdDataCycleTimer, InstanceOfType FB
"LSicar_ProdDataCycleTimer"
   // VAR_INPUT
   //    numberConfigDataSets { ExternalAccessible := 'False'; ExternalVisible := 'False'; ExternalWritable := 'False'} : Int;
   //    dataSetNumber { ExternalAccessible := 'False'; ExternalVisible := 'False'; ExternalWritable := 'False'} : UInt;
   //    pulse100ms { ExternalAccessible := 'False'; ExternalVisible := 'False'; ExternalWritable := 'False'} : Bool;
   // END_VAR
   // VAR_IN_OUT
   //    numberOfDataSets : "LSicar_typeNumberOfDataSets";
   //    dataSet : "LSicar_typeCycleTimer";
   // END_VAR
   // VAR
   //    statCycleTimer { ExternalAccessible := 'False'; ExternalVisible := 'False'; ExternalWritable := 'False'} : Array[0..20] of "LSicar_typeCycleTimerStruct";
   //    statRisEdgeResetAllExt { ExternalAccessible := 'False'; ExternalVisible := 'False'; ExternalWritable := 'False'} : Bool;
   //    statPosPulseResetAllExt { ExternalAccessible := 'False'; ExternalVisible := 'False'; ExternalWritable := 'False'} : Bool;
   //    statRisEdgeResetAll { ExternalAccessible := 'False'; ExternalVisible := 'False'; ExternalWritable := 'False'} : Bool;
   //    statPosPulseResetAll { ExternalAccessible := 'False'; ExternalVisible := 'False'; ExternalWritable := 'False'} : Bool;
   // END_VAR
BEGIN
END_DATA_BLOCK

DATA_BLOCK "InstCycleTimerDataset4"   // DB177
TITLE = Instanz CycleTimerDataset2 / Instance CycleTimerDataset2
{ DB_Accessible_From_OPC_UA := 'FALSE' }
AUTHOR : SICAR
FAMILY : ProdData
// Instanz DB / Instance DB
// stored: DBAccessibleFromOPCUA false, InstanceOfName LSicar_ProdDataCycleTimer, InstanceOfType FB
"LSicar_ProdDataCycleTimer"
   // VAR_INPUT
   //    numberConfigDataSets { ExternalAccessible := 'False'; ExternalVisible := 'False'; ExternalWritable := 'False'} : Int;
   //    dataSetNumber { ExternalAccessible := 'False'; ExternalVisible := 'False'; ExternalWritable := 'False'} : UInt;
   //    pulse100ms { ExternalAccessible := 'False'; ExternalVisible := 'False'; ExternalWritable := 'False'} : Bool;
   // END_VAR
   // VAR_IN_OUT
   //    numberOfDataSets : "LSicar_typeNumberOfDataSets";
   //    dataSet : "LSicar_typeCycleTimer";
   // END_VAR
   // VAR
   //    statCycleTimer { ExternalAccessible := 'False'; ExternalVisible := 'False'; ExternalWritable := 'False'} : Array[0..20] of "LSicar_typeCycleTimerStruct";
   //    statRisEdgeResetAllExt { ExternalAccessible := 'False'; ExternalVisible := 'False'; ExternalWritable := 'False'} : Bool;
   //    statPosPulseResetAllExt { ExternalAccessible := 'False'; ExternalVisible := 'False'; ExternalWritable := 'False'} : Bool;
   //    statRisEdgeResetAll { ExternalAccessible := 'False'; ExternalVisible := 'False'; ExternalWritable := 'False'} : Bool;
   //    statPosPulseResetAll { ExternalAccessible := 'False'; ExternalVisible := 'False'; ExternalWritable := 'False'} : Bool;
   // END_VAR
BEGIN
END_DATA_BLOCK

DATA_BLOCK "InstCycleTimerDataset5"   // DB166
TITLE = Instanz CycleTimerDataset2 / Instance CycleTimerDataset2
{ DB_Accessible_From_OPC_UA := 'FALSE' }
AUTHOR : SICAR
FAMILY : ProdData
// Instanz DB / Instance DB
// stored: DBAccessibleFromOPCUA false, InstanceOfName LSicar_ProdDataCycleTimer, InstanceOfType FB
"LSicar_ProdDataCycleTimer"
   // VAR_INPUT
   //    numberConfigDataSets { ExternalAccessible := 'False'; ExternalVisible := 'False'; ExternalWritable := 'False'} : Int;
   //    dataSetNumber { ExternalAccessible := 'False'; ExternalVisible := 'False'; ExternalWritable := 'False'} : UInt;
   //    pulse100ms { ExternalAccessible := 'False'; ExternalVisible := 'False'; ExternalWritable := 'False'} : Bool;
   // END_VAR
   // VAR_IN_OUT
   //    numberOfDataSets : "LSicar_typeNumberOfDataSets";
   //    dataSet : "LSicar_typeCycleTimer";
   // END_VAR
   // VAR
   //    statCycleTimer { ExternalAccessible := 'False'; ExternalVisible := 'False'; ExternalWritable := 'False'} : Array[0..20] of "LSicar_typeCycleTimerStruct";
   //    statRisEdgeResetAllExt { ExternalAccessible := 'False'; ExternalVisible := 'False'; ExternalWritable := 'False'} : Bool;
   //    statPosPulseResetAllExt { ExternalAccessible := 'False'; ExternalVisible := 'False'; ExternalWritable := 'False'} : Bool;
   //    statRisEdgeResetAll { ExternalAccessible := 'False'; ExternalVisible := 'False'; ExternalWritable := 'False'} : Bool;
   //    statPosPulseResetAll { ExternalAccessible := 'False'; ExternalVisible := 'False'; ExternalWritable := 'False'} : Bool;
   // END_VAR
BEGIN
END_DATA_BLOCK

DATA_BLOCK "InstCycleTimerDataset6"   // DB176
TITLE = Instanz CycleTimerDataset2 / Instance CycleTimerDataset2
{ DB_Accessible_From_OPC_UA := 'FALSE' }
AUTHOR : SICAR
FAMILY : ProdData
// Instanz DB / Instance DB
// stored: DBAccessibleFromOPCUA false, InstanceOfName LSicar_ProdDataCycleTimer, InstanceOfType FB
"LSicar_ProdDataCycleTimer"
   // VAR_INPUT
   //    numberConfigDataSets { ExternalAccessible := 'False'; ExternalVisible := 'False'; ExternalWritable := 'False'} : Int;
   //    dataSetNumber { ExternalAccessible := 'False'; ExternalVisible := 'False'; ExternalWritable := 'False'} : UInt;
   //    pulse100ms { ExternalAccessible := 'False'; ExternalVisible := 'False'; ExternalWritable := 'False'} : Bool;
   // END_VAR
   // VAR_IN_OUT
   //    numberOfDataSets : "LSicar_typeNumberOfDataSets";
   //    dataSet : "LSicar_typeCycleTimer";
   // END_VAR
   // VAR
   //    statCycleTimer { ExternalAccessible := 'False'; ExternalVisible := 'False'; ExternalWritable := 'False'} : Array[0..20] of "LSicar_typeCycleTimerStruct";
   //    statRisEdgeResetAllExt { ExternalAccessible := 'False'; ExternalVisible := 'False'; ExternalWritable := 'False'} : Bool;
   //    statPosPulseResetAllExt { ExternalAccessible := 'False'; ExternalVisible := 'False'; ExternalWritable := 'False'} : Bool;
   //    statRisEdgeResetAll { ExternalAccessible := 'False'; ExternalVisible := 'False'; ExternalWritable := 'False'} : Bool;
   //    statPosPulseResetAll { ExternalAccessible := 'False'; ExternalVisible := 'False'; ExternalWritable := 'False'} : Bool;
   // END_VAR
BEGIN
END_DATA_BLOCK

DATA_BLOCK "InstCycleTimerDataset7"   // DB181
TITLE = Instanz CycleTimerDataset2 / Instance CycleTimerDataset2
{ DB_Accessible_From_OPC_UA := 'FALSE' }
AUTHOR : SICAR
FAMILY : ProdData
// Instanz DB / Instance DB
// stored: DBAccessibleFromOPCUA false, InstanceOfName LSicar_ProdDataCycleTimer, InstanceOfType FB
"LSicar_ProdDataCycleTimer"
   // VAR_INPUT
   //    numberConfigDataSets { ExternalAccessible := 'False'; ExternalVisible := 'False'; ExternalWritable := 'False'} : Int;
   //    dataSetNumber { ExternalAccessible := 'False'; ExternalVisible := 'False'; ExternalWritable := 'False'} : UInt;
   //    pulse100ms { ExternalAccessible := 'False'; ExternalVisible := 'False'; ExternalWritable := 'False'} : Bool;
   // END_VAR
   // VAR_IN_OUT
   //    numberOfDataSets : "LSicar_typeNumberOfDataSets";
   //    dataSet : "LSicar_typeCycleTimer";
   // END_VAR
   // VAR
   //    statCycleTimer { ExternalAccessible := 'False'; ExternalVisible := 'False'; ExternalWritable := 'False'} : Array[0..20] of "LSicar_typeCycleTimerStruct";
   //    statRisEdgeResetAllExt { ExternalAccessible := 'False'; ExternalVisible := 'False'; ExternalWritable := 'False'} : Bool;
   //    statPosPulseResetAllExt { ExternalAccessible := 'False'; ExternalVisible := 'False'; ExternalWritable := 'False'} : Bool;
   //    statRisEdgeResetAll { ExternalAccessible := 'False'; ExternalVisible := 'False'; ExternalWritable := 'False'} : Bool;
   //    statPosPulseResetAll { ExternalAccessible := 'False'; ExternalVisible := 'False'; ExternalWritable := 'False'} : Bool;
   // END_VAR
BEGIN
END_DATA_BLOCK

DATA_BLOCK "InstCycleTimerDataset8"   // DB180
TITLE = Instanz CycleTimerDataset2 / Instance CycleTimerDataset2
{ DB_Accessible_From_OPC_UA := 'FALSE' }
AUTHOR : SICAR
FAMILY : ProdData
// Instanz DB / Instance DB
// stored: DBAccessibleFromOPCUA false, InstanceOfName LSicar_ProdDataCycleTimer, InstanceOfType FB
"LSicar_ProdDataCycleTimer"
   // VAR_INPUT
   //    numberConfigDataSets { ExternalAccessible := 'False'; ExternalVisible := 'False'; ExternalWritable := 'False'} : Int;
   //    dataSetNumber { ExternalAccessible := 'False'; ExternalVisible := 'False'; ExternalWritable := 'False'} : UInt;
   //    pulse100ms { ExternalAccessible := 'False'; ExternalVisible := 'False'; ExternalWritable := 'False'} : Bool;
   // END_VAR
   // VAR_IN_OUT
   //    numberOfDataSets : "LSicar_typeNumberOfDataSets";
   //    dataSet : "LSicar_typeCycleTimer";
   // END_VAR
   // VAR
   //    statCycleTimer { ExternalAccessible := 'False'; ExternalVisible := 'False'; ExternalWritable := 'False'} : Array[0..20] of "LSicar_typeCycleTimerStruct";
   //    statRisEdgeResetAllExt { ExternalAccessible := 'False'; ExternalVisible := 'False'; ExternalWritable := 'False'} : Bool;
   //    statPosPulseResetAllExt { ExternalAccessible := 'False'; ExternalVisible := 'False'; ExternalWritable := 'False'} : Bool;
   //    statRisEdgeResetAll { ExternalAccessible := 'False'; ExternalVisible := 'False'; ExternalWritable := 'False'} : Bool;
   //    statPosPulseResetAll { ExternalAccessible := 'False'; ExternalVisible := 'False'; ExternalWritable := 'False'} : Bool;
   // END_VAR
BEGIN
END_DATA_BLOCK

DATA_BLOCK "InstLimitValueDataset1"   // DB54
TITLE = Instanz LimitValueDataset1 / Instance LimitValueDataset1
{ DB_Accessible_From_OPC_UA := 'FALSE' }
AUTHOR : SICAR
FAMILY : ProdData
// Instanz DB / Instance DB
// stored: DBAccessibleFromOPCUA false, InstanceOfName LSicar_ProdDataLimitValues, InstanceOfType FB
"LSicar_ProdDataLimitValues"
   // VAR_INPUT
   //    numberConfigDataSets { ExternalAccessible := 'False'; ExternalVisible := 'False'; ExternalWritable := 'False'} : Int;
   //    dataSetNumber { ExternalAccessible := 'False'; ExternalVisible := 'False'; ExternalWritable := 'False'} : UInt;
   // END_VAR
   // VAR_IN_OUT
   //    numberOfDataSets : "LSicar_typeNumberOfDataSets";
   //    dataSet : "LSicar_typeLimitValue";
   //    colorCodeSelectButton { ExternalAccessible := 'False'; ExternalVisible := 'False'; ExternalWritable := 'False'} : UInt;
   // END_VAR
   // VAR
   //    statLimitValue { ExternalAccessible := 'False'; ExternalVisible := 'False'; ExternalWritable := 'False'} : Array[0..10] of "LSicar_typeEdgePulseStruct";
   //    statPrewarnActive { ExternalAccessible := 'False'; ExternalVisible := 'False'; ExternalWritable := 'False'} : Bool;
   //    statAlarmActive { ExternalAccessible := 'False'; ExternalVisible := 'False'; ExternalWritable := 'False'} : Bool;
   // END_VAR
BEGIN
END_DATA_BLOCK

DATA_BLOCK "InstLimitValueDataset2"   // DB55
TITLE = Instanz LimitValueDataset2 / Instance LimitValueDataset2
{ DB_Accessible_From_OPC_UA := 'FALSE' }
AUTHOR : SICAR
FAMILY : ProdData
// Instanz DB / Instance DB
// stored: DBAccessibleFromOPCUA false, InstanceOfName LSicar_ProdDataLimitValues, InstanceOfType FB
"LSicar_ProdDataLimitValues"
   // VAR_INPUT
   //    numberConfigDataSets { ExternalAccessible := 'False'; ExternalVisible := 'False'; ExternalWritable := 'False'} : Int;
   //    dataSetNumber { ExternalAccessible := 'False'; ExternalVisible := 'False'; ExternalWritable := 'False'} : UInt;
   // END_VAR
   // VAR_IN_OUT
   //    numberOfDataSets : "LSicar_typeNumberOfDataSets";
   //    dataSet : "LSicar_typeLimitValue";
   //    colorCodeSelectButton { ExternalAccessible := 'False'; ExternalVisible := 'False'; ExternalWritable := 'False'} : UInt;
   // END_VAR
   // VAR
   //    statLimitValue { ExternalAccessible := 'False'; ExternalVisible := 'False'; ExternalWritable := 'False'} : Array[0..10] of "LSicar_typeEdgePulseStruct";
   //    statPrewarnActive { ExternalAccessible := 'False'; ExternalVisible := 'False'; ExternalWritable := 'False'} : Bool;
   //    statAlarmActive { ExternalAccessible := 'False'; ExternalVisible := 'False'; ExternalWritable := 'False'} : Bool;
   // END_VAR
BEGIN
END_DATA_BLOCK

DATA_BLOCK "InstShiftCounterDataset1"   // DB62
TITLE = Instanz ShiftCounterDataset1 / Instance ShiftCounterDataset1
{ DB_Accessible_From_OPC_UA := 'FALSE' }
AUTHOR : SICAR
FAMILY : ProdData
// Instanz DB / Instance DB
// stored: DBAccessibleFromOPCUA false, InstanceOfName LSicar_ProdDataShiftCounter, InstanceOfType FB
"LSicar_ProdDataShiftCounter"
   // VAR_INPUT
   //    numberConfigDataSets { ExternalAccessible := 'False'; ExternalVisible := 'False'; ExternalWritable := 'False'} : Int;
   //    dataSetNumber { ExternalAccessible := 'False'; ExternalVisible := 'False'; ExternalWritable := 'False'} : UInt;
   // END_VAR
   // VAR_IN_OUT
   //    numberOfDataSets : "LSicar_typeNumberOfDataSets";
   //    dataSet : "LSicar_typeShiftCounter";
   // END_VAR
   // VAR
   //    statPartsCurrentCount { ExternalAccessible := 'False'; ExternalVisible := 'False'; ExternalWritable := 'False'} : Array[0..10] of "LSicar_typeEdgePulseStruct";
   //    statRisEdgeResetAllExt { ExternalAccessible := 'False'; ExternalVisible := 'False'; ExternalWritable := 'False'} : Bool;
   //    statPosPulseResetAllExt { ExternalAccessible := 'False'; ExternalVisible := 'False'; ExternalWritable := 'False'} : Bool;
   //    statRisEdgeResetAll { ExternalAccessible := 'False'; ExternalVisible := 'False'; ExternalWritable := 'False'} : Bool;
   //    statPosPulseResetAll { ExternalAccessible := 'False'; ExternalVisible := 'False'; ExternalWritable := 'False'} : Bool;
   // END_VAR
BEGIN
END_DATA_BLOCK

DATA_BLOCK "InstShiftCounterDataset2"   // DB64
TITLE = Instanz ShiftCounterDataset2 / Instance ShiftCounterDataset2
{ DB_Accessible_From_OPC_UA := 'FALSE' }
AUTHOR : SICAR
FAMILY : ProdData
// Instanz DB / Instance DB
// stored: DBAccessibleFromOPCUA false, InstanceOfName LSicar_ProdDataShiftCounter, InstanceOfType FB
"LSicar_ProdDataShiftCounter"
   // VAR_INPUT
   //    numberConfigDataSets { ExternalAccessible := 'False'; ExternalVisible := 'False'; ExternalWritable := 'False'} : Int;
   //    dataSetNumber { ExternalAccessible := 'False'; ExternalVisible := 'False'; ExternalWritable := 'False'} : UInt;
   // END_VAR
   // VAR_IN_OUT
   //    numberOfDataSets : "LSicar_typeNumberOfDataSets";
   //    dataSet : "LSicar_typeShiftCounter";
   // END_VAR
   // VAR
   //    statPartsCurrentCount { ExternalAccessible := 'False'; ExternalVisible := 'False'; ExternalWritable := 'False'} : Array[0..10] of "LSicar_typeEdgePulseStruct";
   //    statRisEdgeResetAllExt { ExternalAccessible := 'False'; ExternalVisible := 'False'; ExternalWritable := 'False'} : Bool;
   //    statPosPulseResetAllExt { ExternalAccessible := 'False'; ExternalVisible := 'False'; ExternalWritable := 'False'} : Bool;
   //    statRisEdgeResetAll { ExternalAccessible := 'False'; ExternalVisible := 'False'; ExternalWritable := 'False'} : Bool;
   //    statPosPulseResetAll { ExternalAccessible := 'False'; ExternalVisible := 'False'; ExternalWritable := 'False'} : Bool;
   // END_VAR
BEGIN
END_DATA_BLOCK

DATA_BLOCK "InstShiftCounterOeeDset1"   // DB124
TITLE = Instanz ShiftCounterOeeDset1 / Instance ShiftCounterOeeDset1
{ DB_Accessible_From_OPC_UA := 'FALSE' }
AUTHOR : SICAR
FAMILY : ProdData
// Instanz DB / Instance DB
// stored: DBAccessibleFromOPCUA false, InstanceOfName LSicar_ProdDataShiftCounterOee, InstanceOfType FB
"LSicar_ProdDataShiftCounterOee"
   // VAR_INPUT
   //    numberConfigDataSets { ExternalAccessible := 'False'; ExternalVisible := 'False'; ExternalWritable := 'False'} : Int;
   //    dataSetNumber { ExternalAccessible := 'False'; ExternalVisible := 'False'; ExternalWritable := 'False'} : UInt;
   //    shiftProdTimeTarget { ExternalAccessible := 'False'; ExternalVisible := 'False'; ExternalWritable := 'False'} : Time;
   //    shiftProdTimeExpired { ExternalAccessible := 'False'; ExternalVisible := 'False'; ExternalWritable := 'False'} : Time;
   // END_VAR
   // VAR_IN_OUT
   //    numberOfDataSets : "LSicar_typeNumberOfDataSets";
   //    dataSet : "LSicar_typeShiftCounterOee";
   // END_VAR
   // VAR
   //    statPartsCurrentCount { ExternalAccessible := 'False'; ExternalVisible := 'False'; ExternalWritable := 'False'} : Array[0..10] of "LSicar_typeEdgePulseStruct";
   //    statPartsCurrentCountOk { ExternalAccessible := 'False'; ExternalVisible := 'False'; ExternalWritable := 'False'} : Array[0..10] of "LSicar_typeEdgePulseStruct";
   //    statFactor { ExternalAccessible := 'False'; ExternalVisible := 'False'; ExternalWritable := 'False'} : "LSicar_typeFactorOee";
   //    statTimeFactorTrend { ExternalAccessible := 'False'; ExternalVisible := 'False'; ExternalWritable := 'False'} : Real;
   //    statShiftProdTimeTarget { ExternalAccessible := 'False'; ExternalVisible := 'False'; ExternalWritable := 'False'} : Real;
   //    statShiftProdTimeExpired { ExternalAccessible := 'False'; ExternalVisible := 'False'; ExternalWritable := 'False'} : Real;
   //    statRisEdgeResetAllExt { ExternalAccessible := 'False'; ExternalVisible := 'False'; ExternalWritable := 'False'} : Bool;
   //    statPosPulseResetAllExt { ExternalAccessible := 'False'; ExternalVisible := 'False'; ExternalWritable := 'False'} : Bool;
   //    statRisEdgeResetAll { ExternalAccessible := 'False'; ExternalVisible := 'False'; ExternalWritable := 'False'} : Bool;
   //    statPosPulseResetAll { ExternalAccessible := 'False'; ExternalVisible := 'False'; ExternalWritable := 'False'} : Bool;
   // END_VAR
BEGIN
END_DATA_BLOCK

DATA_BLOCK "InstShiftCounterOeeDset2"   // DB125
TITLE = Instanz ShiftCounterOeeDset2 / Instance ShiftCounterOeeDset2
{ DB_Accessible_From_OPC_UA := 'FALSE' }
AUTHOR : SICAR
FAMILY : ProdData
// Instanz DB / Instance DB
// stored: DBAccessibleFromOPCUA false, InstanceOfName LSicar_ProdDataShiftCounterOee, InstanceOfType FB
"LSicar_ProdDataShiftCounterOee"
   // VAR_INPUT
   //    numberConfigDataSets { ExternalAccessible := 'False'; ExternalVisible := 'False'; ExternalWritable := 'False'} : Int;
   //    dataSetNumber { ExternalAccessible := 'False'; ExternalVisible := 'False'; ExternalWritable := 'False'} : UInt;
   //    shiftProdTimeTarget { ExternalAccessible := 'False'; ExternalVisible := 'False'; ExternalWritable := 'False'} : Time;
   //    shiftProdTimeExpired { ExternalAccessible := 'False'; ExternalVisible := 'False'; ExternalWritable := 'False'} : Time;
   // END_VAR
   // VAR_IN_OUT
   //    numberOfDataSets : "LSicar_typeNumberOfDataSets";
   //    dataSet : "LSicar_typeShiftCounterOee";
   // END_VAR
   // VAR
   //    statPartsCurrentCount { ExternalAccessible := 'False'; ExternalVisible := 'False'; ExternalWritable := 'False'} : Array[0..10] of "LSicar_typeEdgePulseStruct";
   //    statPartsCurrentCountOk { ExternalAccessible := 'False'; ExternalVisible := 'False'; ExternalWritable := 'False'} : Array[0..10] of "LSicar_typeEdgePulseStruct";
   //    statFactor { ExternalAccessible := 'False'; ExternalVisible := 'False'; ExternalWritable := 'False'} : "LSicar_typeFactorOee";
   //    statTimeFactorTrend { ExternalAccessible := 'False'; ExternalVisible := 'False'; ExternalWritable := 'False'} : Real;
   //    statShiftProdTimeTarget { ExternalAccessible := 'False'; ExternalVisible := 'False'; ExternalWritable := 'False'} : Real;
   //    statShiftProdTimeExpired { ExternalAccessible := 'False'; ExternalVisible := 'False'; ExternalWritable := 'False'} : Real;
   //    statRisEdgeResetAllExt { ExternalAccessible := 'False'; ExternalVisible := 'False'; ExternalWritable := 'False'} : Bool;
   //    statPosPulseResetAllExt { ExternalAccessible := 'False'; ExternalVisible := 'False'; ExternalWritable := 'False'} : Bool;
   //    statRisEdgeResetAll { ExternalAccessible := 'False'; ExternalVisible := 'False'; ExternalWritable := 'False'} : Bool;
   //    statPosPulseResetAll { ExternalAccessible := 'False'; ExternalVisible := 'False'; ExternalWritable := 'False'} : Bool;
   // END_VAR
BEGIN
END_DATA_BLOCK

DATA_BLOCK "InstShiftProductionTimes"   // DB113
TITLE = Instance ShiftProductionTimes
{ DB_Accessible_From_OPC_UA := 'FALSE' }
AUTHOR : SICAR
FAMILY : Shift
// Instance DB
// stored: DBAccessibleFromOPCUA false, InstanceOfName LSicar_ShiftProductionTimes, InstanceOfType FB
"LSicar_ShiftProductionTimes"
   // VAR_OUTPUT
   //    shiftProdTimeTarget { ExternalAccessible := 'False'; ExternalVisible := 'False'; ExternalWritable := 'False'} : Time;
   //    shiftProdTimeExpired { ExternalAccessible := 'False'; ExternalVisible := 'False'; ExternalWritable := 'False'} : Time;
   //    shiftActive { ExternalAccessible := 'False'; ExternalVisible := 'False'; ExternalWritable := 'False'} : Bool;
   //    shiftFinishedPulse { ExternalAccessible := 'False'; ExternalVisible := 'False'; ExternalWritable := 'False'} : Bool;
   // END_VAR
   // VAR_IN_OUT
   //    dateAndTime : "LSicar_typeGlobalDateTime";
   //    prodTimesHmi : "LSicar_typeProdTimesHmi";
   // END_VAR
   // VAR
   //    statCurrShiftTimes { ExternalAccessible := 'False'; ExternalVisible := 'False'; ExternalWritable := 'False'} : "LSicar_typeShiftTimes1Shift";
   //    statActual { ExternalAccessible := 'False'; ExternalVisible := 'False'; ExternalWritable := 'False'} : Time_Of_Day;
   //    statBefore { ExternalAccessible := 'False'; ExternalVisible := 'False'; ExternalWritable := 'False'} : Time_Of_Day;
   //    statDayChange { ExternalAccessible := 'False'; ExternalVisible := 'False'; ExternalWritable := 'False'} : Bool;
   //    statDayChangeSet { ExternalAccessible := 'False'; ExternalVisible := 'False'; ExternalWritable := 'False'} : Bool;
   //    statShift { ExternalAccessible := 'False'; ExternalVisible := 'False'; ExternalWritable := 'False'} : "LSicar_typeShiftmodelInfo";
   //    statProdTimeExpired { ExternalAccessible := 'False'; ExternalVisible := 'False'; ExternalWritable := 'False'} : Time;
   //    statBreak { ExternalAccessible := 'False'; ExternalVisible := 'False'; ExternalWritable := 'False'} : Array[0..4] of "LSicar_typeShiftmodelInfo";
   //    statBreakDurationSummary { ExternalAccessible := 'False'; ExternalVisible := 'False'; ExternalWritable := 'False'} : Time;
   //    statBreakActiveSummary { ExternalAccessible := 'False'; ExternalVisible := 'False'; ExternalWritable := 'False'} : Bool;
   //    statBreakCount { ExternalAccessible := 'False'; ExternalVisible := 'False'; ExternalWritable := 'False'} : USInt;
   //    statProdTimeExpired1 { ExternalAccessible := 'False'; ExternalVisible := 'False'; ExternalWritable := 'False'} : Time;
   //    statProdTimeExpired2 { ExternalAccessible := 'False'; ExternalVisible := 'False'; ExternalWritable := 'False'} : Time;
   //    statFalEdgeShiftActive { ExternalAccessible := 'False'; ExternalVisible := 'False'; ExternalWritable := 'False'} : Bool;
   //    statNegPulseShiftActive { ExternalAccessible := 'False'; ExternalVisible := 'False'; ExternalWritable := 'False'} : Bool;
   // END_VAR
BEGIN
END_DATA_BLOCK

DATA_BLOCK "instAlarmCounter1"   // DB37
// stored: InstanceOfName LER_AlarmCounter, InstanceOfType FB
"LER_AlarmCounter"
   // VAR_INPUT
   //    productionMode : Bool;
   //    countUp : Bool;
   //    countReset : Bool;
   // END_VAR
   // VAR_IN_OUT
   //    hmiInterface : "LER_typeAlarmCounterInterface";
   // END_VAR
   // VAR
   //    statPulse_Up : Bool;
   //    statPulse_Reset : Bool;
   //    statTonTimer : TON_TIME;
   // END_VAR
BEGIN
END_DATA_BLOCK

DATA_BLOCK "instAlarmCounter2"   // DB130
// stored: InstanceOfName LER_AlarmCounter_Sensor, InstanceOfType FB
"LER_AlarmCounter_Sensor"
   // VAR_INPUT
   //    productionMode : Bool;
   //    countUp : Bool;
   //    Sensor : Bool;
   //    detectTime : Time;
   // END_VAR
   // VAR_IN_OUT
   //    hmiInterface : "LER_typeAlarmCounterInterface";
   // END_VAR
   // VAR
   //    statPulse : Bool;
   //    statRisingEdge : Bool;
   //    statTonTimer : TON_TIME;
   //    statSensorOn : TON_TIME;
   //    statSensorOff : TON_TIME;
   // END_VAR
BEGIN
END_DATA_BLOCK

DATA_BLOCK "instAlarmCounter3"   // DB140
// stored: InstanceOfName LER_AlarmCounter_Sensor, InstanceOfType FB
"LER_AlarmCounter_Sensor"
   // VAR_INPUT
   //    productionMode : Bool;
   //    countUp : Bool;
   //    Sensor : Bool;
   //    detectTime : Time;
   // END_VAR
   // VAR_IN_OUT
   //    hmiInterface : "LER_typeAlarmCounterInterface";
   // END_VAR
   // VAR
   //    statPulse : Bool;
   //    statRisingEdge : Bool;
   //    statTonTimer : TON_TIME;
   //    statSensorOn : TON_TIME;
   //    statSensorOff : TON_TIME;
   // END_VAR
BEGIN
END_DATA_BLOCK

DATA_BLOCK "instAlarmCounter4"   // DB187
// stored: InstanceOfName LER_AlarmCounter_Sensor, InstanceOfType FB
"LER_AlarmCounter_Sensor"
   // VAR_INPUT
   //    productionMode : Bool;
   //    countUp : Bool;
   //    Sensor : Bool;
   //    detectTime : Time;
   // END_VAR
   // VAR_IN_OUT
   //    hmiInterface : "LER_typeAlarmCounterInterface";
   // END_VAR
   // VAR
   //    statPulse : Bool;
   //    statRisingEdge : Bool;
   //    statTonTimer : TON_TIME;
   //    statSensorOn : TON_TIME;
   //    statSensorOff : TON_TIME;
   // END_VAR
BEGIN
END_DATA_BLOCK

DATA_BLOCK "instAlarmCounter5"   // DB189
// stored: InstanceOfName LER_AlarmCounter_Sensor, InstanceOfType FB
"LER_AlarmCounter_Sensor"
   // VAR_INPUT
   //    productionMode : Bool;
   //    countUp : Bool;
   //    Sensor : Bool;
   //    detectTime : Time;
   // END_VAR
   // VAR_IN_OUT
   //    hmiInterface : "LER_typeAlarmCounterInterface";
   // END_VAR
   // VAR
   //    statPulse : Bool;
   //    statRisingEdge : Bool;
   //    statTonTimer : TON_TIME;
   //    statSensorOn : TON_TIME;
   //    statSensorOff : TON_TIME;
   // END_VAR
BEGIN
END_DATA_BLOCK

DATA_BLOCK "instAlarmCounter6"   // DB258
// stored: InstanceOfName LER_AlarmCounter_Sensor, InstanceOfType FB
"LER_AlarmCounter_Sensor"
   // VAR_INPUT
   //    productionMode : Bool;
   //    countUp : Bool;
   //    Sensor : Bool;
   //    detectTime : Time;
   // END_VAR
   // VAR_IN_OUT
   //    hmiInterface : "LER_typeAlarmCounterInterface";
   // END_VAR
   // VAR
   //    statPulse : Bool;
   //    statRisingEdge : Bool;
   //    statTonTimer : TON_TIME;
   //    statSensorOn : TON_TIME;
   //    statSensorOff : TON_TIME;
   // END_VAR
BEGIN
END_DATA_BLOCK

DATA_BLOCK "instAlarmCounter7"   // DB259
// stored: InstanceOfName LER_AlarmCounter_Sensor, InstanceOfType FB
"LER_AlarmCounter_Sensor"
   // VAR_INPUT
   //    productionMode : Bool;
   //    countUp : Bool;
   //    Sensor : Bool;
   //    detectTime : Time;
   // END_VAR
   // VAR_IN_OUT
   //    hmiInterface : "LER_typeAlarmCounterInterface";
   // END_VAR
   // VAR
   //    statPulse : Bool;
   //    statRisingEdge : Bool;
   //    statTonTimer : TON_TIME;
   //    statSensorOn : TON_TIME;
   //    statSensorOff : TON_TIME;
   // END_VAR
BEGIN
END_DATA_BLOCK

DATA_BLOCK "instAlarmCounter8"   // DB260
// stored: InstanceOfName LER_AlarmCounter, InstanceOfType FB
"LER_AlarmCounter"
   // VAR_INPUT
   //    productionMode : Bool;
   //    countUp : Bool;
   //    countReset : Bool;
   // END_VAR
   // VAR_IN_OUT
   //    hmiInterface : "LER_typeAlarmCounterInterface";
   // END_VAR
   // VAR
   //    statPulse_Up : Bool;
   //    statPulse_Reset : Bool;
   //    statTonTimer : TON_TIME;
   // END_VAR
BEGIN
END_DATA_BLOCK

DATA_BLOCK "InstShiftmodel"   // DB101
TITLE = Instanz Shiftmodel / InstanceShiftmodel
{ DB_Accessible_From_OPC_UA := 'FALSE' }
AUTHOR : SICAR
FAMILY : Shiftmodel
// Instanz DB / Instance DB
// stored: DBAccessibleFromOPCUA false, InstanceOfName LSicar_Shiftmodel, InstanceOfType FB
"LSicar_Shiftmodel"
   // VAR_OUTPUT
   //    currentShiftCircuitTimes { ExternalAccessible := 'False'; ExternalVisible := 'False'; ExternalWritable := 'False'} : "LSicar_typeShiftmodTime1Shift";
   //    currentShiftTimes { ExternalAccessible := 'False'; ExternalVisible := 'False'; ExternalWritable := 'False'} : "LSicar_typeShiftTimes1Shift";
   // END_VAR
   // VAR_IN_OUT
   //    dateAndTime : "LSicar_typeGlobalDateTime";
   //    shiftTimesHmi : "LSicar_typeShiftmodelHmi";
   //    shiftTimesList : Array[0..10] of "LSicar_typeShiftmodTime1DaySel";
   // END_VAR
   // VAR
   //    statListIdx { ExternalAccessible := 'False'; ExternalVisible := 'False'; ExternalWritable := 'False'} : DInt;
   //    statHmiTimesDay { ExternalAccessible := 'False'; ExternalVisible := 'False'; ExternalWritable := 'False'} : Array[0..7] of "LSicar_typeShiftmodTime1Day";
   //    statHmiSignalsDay { ExternalAccessible := 'False'; ExternalVisible := 'False'; ExternalWritable := 'False'} : Array[0..7] of "LSicar_typeShiftmodSign1Day";
   //    statHmiActualDay { ExternalAccessible := 'False'; ExternalVisible := 'False'; ExternalWritable := 'False'} : USInt;
   //    statShiftTimesListOn { ExternalAccessible := 'False'; ExternalVisible := 'False'; ExternalWritable := 'False'} : Bool;
   //    statSummaryHmi { ExternalAccessible := 'False'; ExternalVisible := 'False'; ExternalWritable := 'False'} : "LSicar_typeShiftmodSumHmi";
   //    statHmiShiftmoListindex { ExternalAccessible := 'False'; ExternalVisible := 'False'; ExternalWritable := 'False'} : USInt;
   //    statZeroDay { ExternalAccessible := 'False'; ExternalVisible := 'False'; ExternalWritable := 'False'} : "LSicar_typeShiftmodTime1Day";
   //    statListIndexOld { ExternalAccessible := 'False'; ExternalVisible := 'False'; ExternalWritable := 'False'} : DInt;
   //    statNumberOfWorkDays { ExternalAccessible := 'False'; ExternalVisible := 'False'; ExternalWritable := 'False'} : USInt;
   //    statTimeOfDayActual { ExternalAccessible := 'False'; ExternalVisible := 'False'; ExternalWritable := 'False'} : Time_Of_Day;
   //    statShiftActual { ExternalAccessible := 'False'; ExternalVisible := 'False'; ExternalWritable := 'False'} : USInt;
   //    statDayCount { ExternalAccessible := 'False'; ExternalVisible := 'False'; ExternalWritable := 'False'} : USInt;
   //    statBreakCount { ExternalAccessible := 'False'; ExternalVisible := 'False'; ExternalWritable := 'False'} : USInt;
   //    statDayChangeNightShift { ExternalAccessible := 'False'; ExternalVisible := 'False'; ExternalWritable := 'False'} : Bool;
   //    statDayChangeCircuitTime { ExternalAccessible := 'False'; ExternalVisible := 'False'; ExternalWritable := 'False'} : Bool;
   //    statCheckCircuitTime { ExternalAccessible := 'False'; ExternalVisible := 'False'; ExternalWritable := 'False'} : "LSicar_typeShiftCircuitTimes";
   //    statRisEdge { ExternalAccessible := 'False'; ExternalVisible := 'False'; ExternalWritable := 'False'} : "LSicar_typeShiftmodSumHmi";
   //    statPosPulse { ExternalAccessible := 'False'; ExternalVisible := 'False'; ExternalWritable := 'False'} : "LSicar_typeShiftmodSumHmi";
   //    statFalEdge { ExternalAccessible := 'False'; ExternalVisible := 'False'; ExternalWritable := 'False'} : "LSicar_typeShiftmodSumHmi";
   //    statNegPulse { ExternalAccessible := 'False'; ExternalVisible := 'False'; ExternalWritable := 'False'} : "LSicar_typeShiftmodSumHmi";
   //    statTimesAndCircuit { ExternalAccessible := 'False'; ExternalVisible := 'False'; ExternalWritable := 'False'} : "LSicar_typeShiftmodTime1Shift";
   //    statOnlyTimes { ExternalAccessible := 'False'; ExternalVisible := 'False'; ExternalWritable := 'False'} : "LSicar_typeShiftTimes1Shift";
   //    statRisEdgeListOn { ExternalAccessible := 'False'; ExternalVisible := 'False'; ExternalWritable := 'False'} : Bool;
   //    statPosPulseListOn { ExternalAccessible := 'False'; ExternalVisible := 'False'; ExternalWritable := 'False'} : Bool;
   //    statFalEdgeListOn { ExternalAccessible := 'False'; ExternalVisible := 'False'; ExternalWritable := 'False'} : Bool;
   //    statNegPulseListOn { ExternalAccessible := 'False'; ExternalVisible := 'False'; ExternalWritable := 'False'} : Bool;
   //    statRisEdgeListChange { ExternalAccessible := 'False'; ExternalVisible := 'False'; ExternalWritable := 'False'} : Bool;
   //    statPosPulseListChange { ExternalAccessible := 'False'; ExternalVisible := 'False'; ExternalWritable := 'False'} : Bool;
   //    statFirstCycle { ExternalAccessible := 'False'; ExternalVisible := 'False'; ExternalWritable := 'False'} : Bool;
   // END_VAR
BEGIN
END_DATA_BLOCK

DATA_BLOCK "EeMonitor"   // DB61
TITLE = EeMonitor
AUTHOR : SICAR
FAMILY : DB
// Globale EEM Informationen / Global EEM Information
// stored: InstanceOfName LSicar_typeEemDataHmi, InstanceOfType UDT
"LSicar_typeEemDataHmi"
   // VAR
   //    measurePointIndex : USInt;
   //    measConfiguration { ExternalWritable := 'False'} : EnS_EEm_typeMeasConfig;
   //    measOperationHmi { ExternalWritable := 'False'} : EnS_EEm_typeMeasOperation;
   //    work { ExternalWritable := 'False'} : "LSicar_typeEnMeterWorkHmi";
   // END_VAR
BEGIN
END_DATA_BLOCK

DATA_BLOCK "EeMonitorData"   // DB108
TITLE = EeMonitorData
AUTHOR : SICAR
FAMILY : DB
// Energy efficency monitor Daten / Energy efficency monitor data
// stored: InstanceOfName LSicar_typeEemData, InstanceOfType UDT
"LSicar_typeEemData"
   // VAR
   //    machineConfiguration : EnS_EEm_typeConfig;
   //    machineOperation : EnS_EEm_typeOperation;
   //    measConfiguration : Array[0..9] of EnS_EEm_typeMeasConfig;
   //    measOperation : Array[0..9] of EnS_EEm_typeMeasOperation;
   //    internalData : "LSicar_typeEemDataInternal";
   //    calcError : Bool;
   //    calcStatus : Word;
   //    calcRetVal : Int;
   //    reportCreateCsv : Bool;
   //    reportStatus : Word;
   //    reportNameCsv : String[80];
   // END_VAR
BEGIN
   machineConfiguration.eStateName[1] := 'Auto';
   machineConfiguration.eStateName[2] := 'Auto Preselect';
   machineConfiguration.eStateName[3] := 'Manual';
   machineConfiguration.eStateName[4] := 'Idle';
   machineConfiguration.eStateName[5] := 'Fault';
   machineConfiguration.eStateName[6..7] := '-Not used-';
   machineOperation.maskEnPI := 16#0002;
   measConfiguration[2]."name" := 'PAC Electrical Infeed';
   measConfiguration[3..9]."name" := 'MeasPointXX';
   measConfiguration[2].nameShort := 'P01';
   measConfiguration[3..9].nameShort := 'XX01';
   measConfiguration[2..9].media := 'electrical';
   measConfiguration[2..9].unitCounterNumber := 1;
   measConfiguration[2..9].unitCounterText := 'Wh';
   measConfiguration[2..9].unitActValueNumber := 0;
   measConfiguration[2..9].unitActValueText := 'W';
   measConfiguration[2..9].inputType := 1;
   measConfiguration[2..9].type1Counter.overflowCntValue := 1000000.0;
   measConfiguration[2..9].type1Counter.normFactor := 1.0;
   internalData.productiveEnergyStates[1] := true;
END_DATA_BLOCK

DATA_BLOCK "InstE2MenergyMeterDriver"   // DB56
TITLE = Instanz von FB E2MenergyMeterDrv / Instance of FB E2MenergyMeterDrv
AUTHOR : SICAR
FAMILY : E2M
NAME : E2M_AIEM
VERSION : 2.0
// Energy Meter
// stored: InstanceOfName E2MenergyMeterDrv, InstanceOfType FB
"E2MenergyMeterDrv"
   // VAR_INPUT
   //    id : HW_IO;
   //    firstByteData : Int;
   //    connectionType : Int;
   //    commResourceLimit : Int;
   //    automaticUpdate : Bool;
   //    resetMinMax : Bool;
   //    resetEnergyCounter : Bool;
   //    bitsConnectedHmi : Bool;
   //    backupCycleEnCount : Time;
   // END_VAR
   // VAR_OUTPUT
   //    timeBetweenUpdate : Time;
   //    timeBetweenUpdateMax : Time;
   //    timeStampMeasValues : DTL;
   //    driverData { ExternalAccessible := 'False'; ExternalVisible := 'False'; ExternalWritable := 'False'} : "LSicar_typeEnMeterVisuStruct";
   //    energyCounter { ExternalAccessible := 'False'; ExternalVisible := 'False'; ExternalWritable := 'False'} : "typeEnCounter";
   //    errorCode : DWord;
   //    errorLocation : Word;
   //    timeStampEnCount : DTL;
   // END_VAR
   // VAR_IN_OUT
   //    bitsHmi : "typeEnMeterBits";
   //    commResourceCounter : Int;
   // END_VAR
   // VAR
   //    instReadDataRecord { S7_SetPoint := 'True'} : RDREC;
   //    instWriteDataRecord { S7_SetPoint := 'True'} : WRREC;
   //    instEnCountUpdateTimer { S7_SetPoint := 'True'} : TON_TIME;
   //    instTimeMeasurement { S7_SetPoint := 'True'} : TON_TIME;
   //    instWatchdog { S7_SetPoint := 'True'} : TON_TIME;
   //    statInputVariablesOk : Bool;
   //    statResetEnCountRequest : Bool;
   //    statReadDataRecRequest : Bool;
   //    statWriteDataRecRequest : Bool;
   //    statRestoreEnergy : Bool;
   //    statStartAcyclicHmiOld : Bool;
   //    statResetEnergyHmiOld : Bool;
   //    statResetEnergyOld : Bool;
   //    statResetMinMaxHmiOld : Bool;
   //    statResetMinMaxOld : Bool;
   //    statRunUpdateTimer : Bool;
   //    statWatchdogRun : Bool;
   //    statUserDataVariant : Byte;
   //    statSmState : Int;
   //    statSmStateNext : Int;
   //    statReadRecIndex : Int;
   //    statReadRecMaxLength : UInt;
   //    statTimetoUpdate : Time;
   //    statVmeasurementValues : "typeEnMeterValues";
   //    statVenergyCounter : "typeEnMeterCounter";
   //    statBitsInternalHmi : "typeEnMeterBits";
   // END_VAR
   // VAR RETAIN
   //    statRestoreEnCountValues : "typeEnMeterRestore";
   // END_VAR
   // VAR
   //    statAuxTimeBetweenUpdateMax { S7_SetPoint := 'True'} : Time;
   //    statErrorCode { ExternalVisible := 'False'} : DWord;
   // END_VAR
BEGIN
END_DATA_BLOCK

DATA_BLOCK "InstEmDataHmi"   // DB44
TITLE = Instanz von FB EnergyMeterDataToHmi / Instance of FB instance of FB EnergyMeterDataToHmi
AUTHOR : SICAR
FAMILY : Energy
VERSION : 1.0
// Energy meter HMI
// stored: InstanceOfName LSicar_EnMeterDataToHmi, InstanceOfType FB
"LSicar_EnMeterDataToHmi"
   // VAR_INPUT
   //    energyMeter01Visu { ExternalAccessible := 'False'; ExternalVisible := 'False'; ExternalWritable := 'False'} : "LSicar_typeEnMeterVisuStruct";
   //    energyMeter02Visu { ExternalAccessible := 'False'; ExternalVisible := 'False'; ExternalWritable := 'False'} : "LSicar_typeEnMeterVisuStruct";
   //    energyMeter03Visu { ExternalAccessible := 'False'; ExternalVisible := 'False'; ExternalWritable := 'False'} : "LSicar_typeEnMeterVisuStruct";
   //    energyMeter04Visu { ExternalAccessible := 'False'; ExternalVisible := 'False'; ExternalWritable := 'False'} : "LSicar_typeEnMeterVisuStruct";
   //    energyMeter05Visu { ExternalAccessible := 'False'; ExternalVisible := 'False'; ExternalWritable := 'False'} : "LSicar_typeEnMeterVisuStruct";
   //    energyMeter06Visu { ExternalAccessible := 'False'; ExternalVisible := 'False'; ExternalWritable := 'False'} : "LSicar_typeEnMeterVisuStruct";
   //    energyMeter07Visu { ExternalAccessible := 'False'; ExternalVisible := 'False'; ExternalWritable := 'False'} : "LSicar_typeEnMeterVisuStruct";
   //    energyMeter08Visu { ExternalAccessible := 'False'; ExternalVisible := 'False'; ExternalWritable := 'False'} : "LSicar_typeEnMeterVisuStruct";
   // END_VAR
   // VAR
   //    statEmIndex : Int;
   //    statEmData : "LSicar_typeEnMeterVisuStruct";
   //    statResetMinMaxAll : Bool;
   //    statResetMinMax : Array[0..8] of Bool;
   //    statResetEnCounterAll : Bool;
   //    statResetEnCounter : Array[0..8] of Bool;
   // END_VAR
BEGIN
END_DATA_BLOCK

DATA_BLOCK "InstPlantSimulationTimer"   // DB110
{ DB_Accessible_From_OPC_UA := 'FALSE' }
// stored: DBAccessibleFromOPCUA false, DBAccessibleFromWebserver false, InstanceOfName IEC_TIMER, OfSystemLibElement IEC_TIMER, OfSystemLibVersion 1.0
"IEC_TIMER"
   // VAR
   //    PT : Time;
   //    ET { ExternalWritable := 'False'} : Time;
   //    IN : Bool;
   //    Q { ExternalWritable := 'False'} : Bool;
   // END_VAR
BEGIN
END_DATA_BLOCK

DATA_BLOCK "InstSimulationTimer"   // DB111
TITLE = Simulation timer
// Instanz of IEC timer / instance of IEC timer
// stored: InstanceOfName IEC_TIMER, OfSystemLibElement IEC_TIMER, OfSystemLibVersion 1.0
"IEC_TIMER"
   // VAR
   //    PT : Time;
   //    ET { ExternalWritable := 'False'} : Time;
   //    IN : Bool;
   //    Q { ExternalWritable := 'False'} : Bool;
   // END_VAR
BEGIN
END_DATA_BLOCK

DATA_BLOCK "InstSleepModeManager"   // DB293
// stored: InstanceOfName LER_SleepModeManager, InstanceOfType FB
"LER_SleepModeManager"
   // VAR_INPUT
   //    enable : Bool;
   //    unitStatus : "LAF_typeUnitStatus";
   //    wakeUpReq : Bool;
   //    sleepDelay : Time;
   //    deepSleepDelay : Time;
   // END_VAR
   // VAR_OUTPUT
   //    sleepModeChangeReq : Bool;
   //    deepSleepModeChangeReq : Bool;
   //    wakeUpRecoveryRequired : Bool;
   // END_VAR
   // VAR
   //    instSleepDelay { ExternalAccessible := 'False'; ExternalVisible := 'False'; ExternalWritable := 'False'; S7_SetPoint := 'True'} : TON_TIME;
   //    instDeepSleepDelay { ExternalAccessible := 'False'; ExternalVisible := 'False'; ExternalWritable := 'False'; S7_SetPoint := 'True'} : TON_TIME;
   //    statStandbyReady { ExternalAccessible := 'False'; ExternalVisible := 'False'; ExternalWritable := 'False'} : Bool;
   //    statWakeUpRecoveryRequired { ExternalAccessible := 'False'; ExternalVisible := 'False'; ExternalWritable := 'False'} : Bool;
   // END_VAR
BEGIN
END_DATA_BLOCK

DATA_BLOCK "InstChecksum"   // DB50
AUTHOR : SICAR
FAMILY : Diag
// stored: AssignedProDiagFB ProDiag, InstanceOfName LAF_Checksum, InstanceOfType FB
"LAF_Checksum"
   // VAR_INPUT
   //    plantIdentifier { ExternalAccessible := 'False'; ExternalVisible := 'False'; ExternalWritable := 'False'} : WString[24];
   //    textListId { ExternalAccessible := 'False'; ExternalVisible := 'False'; ExternalWritable := 'False'} : Int;
   //    dateTime { ExternalAccessible := 'False'; ExternalVisible := 'False'; ExternalWritable := 'False'} : Date_And_Time;
   //    readChecksum { ExternalAccessible := 'False'; ExternalVisible := 'False'; ExternalWritable := 'False'} : Bool;
   //    ack { ExternalAccessible := 'False'; ExternalVisible := 'False'; ExternalWritable := 'False'} : Bool;
   //    hideMessageStandard { ExternalAccessible := 'False'; ExternalVisible := 'False'; ExternalWritable := 'False'} : Bool;
   //    hideMessageSafety { ExternalAccessible := 'False'; ExternalVisible := 'False'; ExternalWritable := 'False'} : Bool;
   //    hideMessageTextlist { ExternalAccessible := 'False'; ExternalVisible := 'False'; ExternalWritable := 'False'} : Bool;
   // END_VAR
   // VAR_OUTPUT
   //    generalMessage { ExternalAccessible := 'False'; ExternalVisible := 'False'; ExternalWritable := 'False'} : Bool;
   // END_VAR
   // VAR_IN_OUT
   //    checksumHmi : "LAF_typeChecksum";
   // END_VAR
   // VAR
   //    statReadChecksumStorage { ExternalAccessible := 'False'; ExternalVisible := 'False'; ExternalWritable := 'False'} : Bool;
   //    statChecksumStandard { ExternalAccessible := 'False'; ExternalVisible := 'False'; ExternalWritable := 'False'} : Array[0..7] of Byte;
   //    statChecksumStafety { ExternalAccessible := 'False'; ExternalVisible := 'False'; ExternalWritable := 'False'} : Array[0..7] of Byte;
   //    statChecksumTextlists { ExternalAccessible := 'False'; ExternalVisible := 'False'; ExternalWritable := 'False'} : Array[0..7] of Byte;
   //    statChecksumStandOldNull { ExternalAccessible := 'False'; ExternalVisible := 'False'; ExternalWritable := 'False'} : Bool;
   //    statChecksumSafeOldNull { ExternalAccessible := 'False'; ExternalVisible := 'False'; ExternalWritable := 'False'} : Bool;
   //    statChecksumTextlOldNull { ExternalAccessible := 'False'; ExternalVisible := 'False'; ExternalWritable := 'False'} : Bool;
   //    statChecksumStandDiff { ExternalAccessible := 'False'; ExternalVisible := 'False'; ExternalWritable := 'False'} : Bool;
   //    statChecksumSafeDiff { ExternalAccessible := 'False'; ExternalVisible := 'False'; ExternalWritable := 'False'} : Bool;
   //    statChecksumTextlDiff { ExternalAccessible := 'False'; ExternalVisible := 'False'; ExternalWritable := 'False'} : Bool;
   //    instGetChecksum1 { ExternalAccessible := 'False'; ExternalVisible := 'False'; ExternalWritable := 'False'} : GetChecksum;
   //    instGetChecksum2 { ExternalAccessible := 'False'; ExternalVisible := 'False'; ExternalWritable := 'False'} : GetChecksum;
   //    instGetChecksum3 { ExternalAccessible := 'False'; ExternalVisible := 'False'; ExternalWritable := 'False'} : GetChecksum;
   //    statRetValHta { ExternalAccessible := 'False'; ExternalVisible := 'False'; ExternalWritable := 'False'} : "LAF_typeChecksumCatWord";
   //    statRisEdgeDiff { ExternalAccessible := 'False'; ExternalVisible := 'False'; ExternalWritable := 'False'} : "LAF_typeChecksumCatBool";
   //    statMessageStandModified { ExternalAccessible := 'False'; ExternalVisible := 'False'; ExternalWritable := 'False'} : Bool;
   //    statMessageSafeModified { ExternalAccessible := 'False'; ExternalVisible := 'False'; ExternalWritable := 'False'} : Bool;
   //    statMessageTextlModified { ExternalAccessible := 'False'; ExternalVisible := 'False'; ExternalWritable := 'False'} : Bool;
   //    statWarnNoStandard { ExternalAccessible := 'False'; ExternalVisible := 'False'; ExternalWritable := 'False'} : UInt;
   //    statWarnNoSafety { ExternalAccessible := 'False'; ExternalVisible := 'False'; ExternalWritable := 'False'} : UInt;
   //    statWarnNoTextlist { ExternalAccessible := 'False'; ExternalVisible := 'False'; ExternalWritable := 'False'} : UInt;
   // END_VAR
BEGIN
END_DATA_BLOCK

DATA_BLOCK "InstMemCardDiag"   // DB122
AUTHOR : Siemens Digital Industries
FAMILY : LAF
// stored: AssignedProDiagFB ProDiag, InstanceOfName LAF_MemCardDiag, InstanceOfType FB
"LAF_MemCardDiag"
   // VAR_INPUT
   //    plantIdentifier { ExternalAccessible := 'False'; ExternalVisible := 'False'; ExternalWritable := 'False'} : WString[24];
   //    textListId { ExternalAccessible := 'False'; ExternalVisible := 'False'; ExternalWritable := 'False'} : Int;
   //    firstCycle { ExternalAccessible := 'False'; ExternalVisible := 'False'; ExternalWritable := 'False'} : Bool;
   //    readInfoMemCard { ExternalAccessible := 'False'; ExternalVisible := 'False'; ExternalWritable := 'False'} : Bool;
   //    hideAlarmMask { ExternalAccessible := 'False'; ExternalVisible := 'False'; ExternalWritable := 'False'} : Byte;
   // END_VAR
   // VAR_OUTPUT
   //    generalAlarm { ExternalAccessible := 'False'; ExternalVisible := 'False'; ExternalWritable := 'False'} : Bool;
   //    generalWarn { ExternalAccessible := 'False'; ExternalVisible := 'False'; ExternalWritable := 'False'} : Bool;
   //    generalInfo { ExternalAccessible := 'False'; ExternalVisible := 'False'; ExternalWritable := 'False'} : Bool;
   // END_VAR
   // VAR_IN_OUT
   //    diagHmi : "LAF_typeMemCardDiag";
   // END_VAR
   // VAR
   //    statMessages { ExternalAccessible := 'False'; ExternalVisible := 'False'; ExternalWritable := 'False'} : "LAF_typeMemCardMessages";
   //    statHideMessages { ExternalAccessible := 'False'; ExternalVisible := 'False'; ExternalWritable := 'False'} : "LAF_typeMemCardMessages";
   //    statStep { ExternalAccessible := 'False'; ExternalVisible := 'False'; ExternalWritable := 'False'} : Array[0..3] of Bool;
   //    statRisEdgeStep0 { ExternalAccessible := 'False'; ExternalVisible := 'False'; ExternalWritable := 'False'} : Bool;
   //    statRisEdgeStep1 { ExternalAccessible := 'False'; ExternalVisible := 'False'; ExternalWritable := 'False'} : Bool;
   //    statAlarmNo { ExternalAccessible := 'False'; ExternalVisible := 'False'; ExternalWritable := 'False'} : UInt;
   //    statWarnNo { ExternalAccessible := 'False'; ExternalVisible := 'False'; ExternalWritable := 'False'} : UInt;
   //    statInfoNo { ExternalAccessible := 'False'; ExternalVisible := 'False'; ExternalWritable := 'False'} : UInt;
   //    instGetInfoMode0 { ExternalAccessible := 'False'; ExternalVisible := 'False'; ExternalWritable := 'False'} : GetSMCinfo;
   //    instGetInfoMode1 { ExternalAccessible := 'False'; ExternalVisible := 'False'; ExternalWritable := 'False'} : GetSMCinfo;
   //    instGetInfoMode2 { ExternalAccessible := 'False'; ExternalVisible := 'False'; ExternalWritable := 'False'} : GetSMCinfo;
   //    instGetInfoMode3 { ExternalAccessible := 'False'; ExternalVisible := 'False'; ExternalWritable := 'False'} : GetSMCinfo;
   // END_VAR
BEGIN
END_DATA_BLOCK

DATA_BLOCK "InstPlcDiag"   // DB42
AUTHOR : Siemens Digital Industries
FAMILY : LAF
// stored: InstanceOfName LAF_PlcDiag, InstanceOfType FB
"LAF_PlcDiag"
   // VAR_INPUT
   //    localCommon { ExternalAccessible := 'False'; ExternalVisible := 'False'; ExternalWritable := 'False'} : HW_SUBMODULE;
   //    localProfinetInterface { ExternalAccessible := 'False'; ExternalVisible := 'False'; ExternalWritable := 'False'} : HW_INTERFACE;
   //    firstCycle { ExternalAccessible := 'False'; ExternalVisible := 'False'; ExternalWritable := 'False'} : Bool;
   // END_VAR
   // VAR_IN_OUT
   //    diagDataHmi : "LAF_typePlcDiag";
   // END_VAR
   // VAR
   //    statLocalCommon { ExternalAccessible := 'False'; ExternalVisible := 'False'; ExternalWritable := 'False'} : HW_SUBMODULE;
   //    statLocProfinetInterface { ExternalAccessible := 'False'; ExternalVisible := 'False'; ExternalWritable := 'False'} : HW_INTERFACE;
   //    instGetImData0 { ExternalAccessible := 'False'; ExternalVisible := 'False'; ExternalWritable := 'False'} : Get_IM_Data;
   //    statGetImData0ErrorSaved { ExternalAccessible := 'False'; ExternalVisible := 'False'; ExternalWritable := 'False'} : Word;
   //    instGetImData1 { ExternalAccessible := 'False'; ExternalVisible := 'False'; ExternalWritable := 'False'} : Get_IM_Data;
   //    statGetImData1ErrorSaved { ExternalAccessible := 'False'; ExternalVisible := 'False'; ExternalWritable := 'False'} : Word;
   //    instGetImData2 { ExternalAccessible := 'False'; ExternalVisible := 'False'; ExternalWritable := 'False'} : Get_IM_Data;
   //    statGetImData2ErrorSaved { ExternalAccessible := 'False'; ExternalVisible := 'False'; ExternalWritable := 'False'} : Word;
   //    instGetImData3 { ExternalAccessible := 'False'; ExternalVisible := 'False'; ExternalWritable := 'False'} : Get_IM_Data;
   //    statGetImData3ErroSaved { ExternalAccessible := 'False'; ExternalVisible := 'False'; ExternalWritable := 'False'} : Word;
   //    instReadRecord { ExternalAccessible := 'False'; ExternalVisible := 'False'; ExternalWritable := 'False'} : RDREC;
   //    statReadRecordResult { ExternalAccessible := 'False'; ExternalVisible := 'False'; ExternalWritable := 'False'} : Array[0..199] of Byte;
   //    statStartNetAddresses { ExternalAccessible := 'False'; ExternalVisible := 'False'; ExternalWritable := 'False'} : USInt;
   //    statIm1PlDesiLocIdLen { ExternalAccessible := 'False'; ExternalVisible := 'False'; ExternalWritable := 'False'} : Int;
   //    statRisEdgeReadAll { ExternalAccessible := 'False'; ExternalVisible := 'False'; ExternalWritable := 'False'} : Bool;
   //    statPosPulseReadAll { ExternalAccessible := 'False'; ExternalVisible := 'False'; ExternalWritable := 'False'} : Bool;
   //    statErrorText { ExternalAccessible := 'False'; ExternalVisible := 'False'; ExternalWritable := 'False'} : String[30];
   // END_VAR
BEGIN
END_DATA_BLOCK

DATA_BLOCK "IdentRfInterfaceHmi"   // DB218
// stored: InstanceOfName typeIdentRfHmi, InstanceOfType UDT
"typeIdentRfHmi"
BEGIN
END_DATA_BLOCK

DATA_BLOCK "instGetIdentRf"   // DB165
// stored: InstanceOfName GetIdentRf, InstanceOfType FB
"GetIdentRf"
BEGIN
END_DATA_BLOCK

DATA_BLOCK "instRfidAntenaLeft"   // DB67
// stored: AssignedProDiagFB ProDiag, InstanceOfName LER_RFID, InstanceOfType FB
"LER_RFID"
   // VAR_INPUT
   //    enable : Bool;
   //    enableManualCmds : Bool;
   //    bobinChuck : Bool;
   // END_VAR
   // VAR_OUTPUT
   //    error : Bool;
   //    status : DWord;
   // END_VAR
   // VAR_IN_OUT
   //    RFID_Chanel : TO_IDENT;
   //    IdentRfAntena : "LSicar_typeIdentInterfaceHmi";
   //    moduleInterface : "LER_typeRFIDInterface";
   // END_VAR
   // VAR
   //    instResetReader : Reset_Reader;
   //    instRead : Read;
   //    instWrite : Write;
   //    instInventory : Inventory;
   //    statResetReaderUDT : "LER_typeResetReaderUDT";
   //    statReadUDT : "LER_typeReadWriteUDT";
   //    statWriteUDT : "LER_typeReadWriteUDT";
   //    statInventoryUDT : "LER_typeInventoryUDT";
   //    statResultRFIDReset : Bool;
   //    statPulse : Array[0..9] of Bool;
   //    statTonTimer : TON_TIME;
   //    statBobinData : IID_IN_I_81;
   //    statRFID_str : String[32];
   //    statEPCID_str : String[32];
   //    statHi : Byte;
   //    statLo : Byte;
   //    statHexArray : Array[0..15] of Char;
   // END_VAR
BEGIN
END_DATA_BLOCK

DATA_BLOCK "instRfidAntenaRight"   // DB167
// stored: AssignedProDiagFB ProDiag, InstanceOfName LER_RFID, InstanceOfType FB
"LER_RFID"
   // VAR_INPUT
   //    enable : Bool;
   //    enableManualCmds : Bool;
   //    bobinChuck : Bool;
   // END_VAR
   // VAR_OUTPUT
   //    error : Bool;
   //    status : DWord;
   // END_VAR
   // VAR_IN_OUT
   //    RFID_Chanel : TO_IDENT;
   //    IdentRfAntena : "LSicar_typeIdentInterfaceHmi";
   //    moduleInterface : "LER_typeRFIDInterface";
   // END_VAR
   // VAR
   //    instResetReader : Reset_Reader;
   //    instRead : Read;
   //    instWrite : Write;
   //    instInventory : Inventory;
   //    statResetReaderUDT : "LER_typeResetReaderUDT";
   //    statReadUDT : "LER_typeReadWriteUDT";
   //    statWriteUDT : "LER_typeReadWriteUDT";
   //    statInventoryUDT : "LER_typeInventoryUDT";
   //    statResultRFIDReset : Bool;
   //    statPulse : Array[0..9] of Bool;
   //    statTonTimer : TON_TIME;
   //    statBobinData : IID_IN_I_81;
   //    statRFID_str : String[32];
   //    statEPCID_str : String[32];
   //    statHi : Byte;
   //    statLo : Byte;
   //    statHexArray : Array[0..15] of Char;
   // END_VAR
BEGIN
END_DATA_BLOCK

DATA_BLOCK "instRfidMobile"   // DB283
// stored: InstanceOfName LER_RFID_Mobile, InstanceOfType FB
"LER_RFID_Mobile"
   // VAR_INPUT
   //    enable : Bool;
   //    enableManualCmds : Bool;
   // END_VAR
   // VAR_OUTPUT
   //    error : Bool;
   //    status : DWord;
   // END_VAR
   // VAR_IN_OUT
   //    IdentRfAntena : "LSicar_typeIdentInterfaceHmi";
   //    moduleInterface : "LER_typeMobileRFIDInterface";
   // END_VAR
   // VAR
   //    instTRCV_C : TRCV_C;
   //    statConnectionData : TCON_IP_v4;
   //    statTrcvUDT : "LER_typeTrcvUDT";
   //    statResultRFIDReset : Bool;
   //    statPulse : Array[0..9] of Bool;
   //    statTonTimer : TON_TIME;
   //    statBobinData : IID_IN_I_81;
   //    statRFID_str : String[32];
   //    statEPCID_str : String[32];
   //    statHi : Byte;
   //    statLo : Byte;
   //    statHexArray : Array[0..15] of Char;
   // END_VAR
BEGIN
END_DATA_BLOCK
